LIN {X 0,Y 205.064,Z 329.408,A -85,B 0,C 180,E1 -21802.532,E2 -21802.532} C_VEL
LIN {X 0,Y 207.762,Z 331.827,A -85,B 0,C 180,E1 -21804.481,E2 -21804.481} C_VEL
LIN {X 0,Y 210.172,Z 335.291,A -85,B 0,C 180,E1 -21806.167,E2 -21806.167} C_VEL
LIN {X 0,Y 211.843,Z 337.01,A -85,B 0,C 180,E1 -21807.207,E2 -21807.207} C_VEL
LIN {X 0,Y 214.618,Z 340.729,A -85,B 0,C 180,E1 -21808.883,E2 -21808.883} C_VEL
LIN {X 0,Y 216.211,Z 342.811,A -85,B 0,C 180,E1 -21809.784,E2 -21809.784} C_VEL
LIN {X 0,Y 219.819,Z 347.623,A -85,B 0,C 180,E1 -21811.698,E2 -21811.698} C_VEL
LIN {X 0,Y 224.599,Z 354.224,A -85,B 0,C 180,E1 -21814.01,E2 -21814.01} C_VEL
LIN {X 0,Y 231.76,Z 365.241,A -85,B 0,C 180,E1 -21817.132,E2 -21817.132} C_VEL
LIN {X 0,Y 239.139,Z 377.762,A -85,B 0,C 180,E1 -21820.005,E2 -21820.005} C_VEL
LIN {X 0,Y 243.057,Z 385.535,A -85,B 0,C 180,E1 -21821.444,E2 -21821.444} C_VEL
LIN {X 0,Y 244.176,Z 388.149,A -85,B 0,C 180,E1 -21821.856,E2 -21821.856} C_VEL
LIN {X 0,Y 238.992,Z 467.481,A -85,B 0,C 180,E1 -21823.985,E2 -21823.985} C_VEL
LIN {X 0,Y 237.015,Z 483.086,A -85,B 0,C 180,E1 -21824.632,E2 -21824.632} C_VEL
LIN {X 0,Y 234.342,Z 498.666,A -85,B 0,C 180,E1 -21825.643,E2 -21825.643} C_VEL
LIN {X 0,Y 230.951,Z 513.459,A -85,B 0,C 180,E1 -21826.943,E2 -21826.943} C_VEL
LIN {X 0,Y 227.125,Z 527.553,A -85,B 0,C 180,E1 -21828.594,E2 -21828.594} C_VEL
LIN {X 0,Y 222.938,Z 539.758,A -85,B 0,C 180,E1 -21830.331,E2 -21830.331} C_VEL
LIN {X 0,Y 218.747,Z 551.094,A -85,B 0,C 180,E1 -21832.38,E2 -21832.38} C_VEL
LIN {X 0,Y 213.85,Z 562.546,A -85,B 0,C 180,E1 -21834.893,E2 -21834.893} C_VEL
LIN {X 0,Y 210.165,Z 571.106,A -85,B 0,C 180,E1 -21837.245,E2 -21837.245} C_VEL
LIN {X 0,Y 205.664,Z 580.387,A -85,B 0,C 180,E1 -21840.298,E2 -21840.298} C_VEL
LIN {X 0,Y 201.657,Z 588.46,A -85,B 0,C 180,E1 -21843.619,E2 -21843.619} C_VEL
LIN {X 0,Y 197.889,Z 595.794,A -85,B 0,C 180,E1 -21847.427,E2 -21847.427} C_VEL
LIN {X 0,Y 195.175,Z 601.274,A -85,B 0,C 180,E1 -21851.091,E2 -21851.091} C_VEL
LIN {X 0,Y 192.884,Z 606.023,A -85,B 0,C 180,E1 -21855.224,E2 -21855.224} C_VEL
LIN {X 0,Y 191.454,Z 609.492,A -85,B 0,C 180,E1 -21859.424,E2 -21859.424} C_VEL
LIN {X 0,Y 190.598,Z 611.782,A -85,B 0,C 180,E1 -21863.649,E2 -21863.649} C_VEL
LIN {X 0,Y 190.279,Z 612.946,A -85,B 0,C 180,E1 -21867.883,E2 -21867.883} C_VEL
LIN {X 0,Y 190.301,Z 613.099,A -85,B 0,C 180,E1 -21870,E2 -21870} C_VEL
LIN {X 0,Y 190.444,Z 612.387,A -85,B 0,C 180,E1 -21874.869,E2 -21874.869} C_VEL
LIN {X 0,Y 190.924,Z 610.864,A -85,B 0,C 180,E1 -21878.467,E2 -21878.467} C_VEL
LIN {X 0,Y 192.015,Z 608.037,A -85,B 0,C 180,E1 -21882.686,E2 -21882.686} C_VEL
LIN {X 0,Y 193.838,Z 603.984,A -85,B 0,C 180,E1 -21886.861,E2 -21886.861} C_VEL
LIN {X 0,Y 196.543,Z 598.603,A -85,B 0,C 180,E1 -21890.951,E2 -21890.951} C_VEL
LIN {X 0,Y 199.996,Z 591.742,A -85,B 0,C 180,E1 -21894.941,E2 -21894.941} C_VEL
LIN {X 0,Y 204.381,Z 583.169,A -85,B 0,C 180,E1 -21898.777,E2 -21898.777} C_VEL
LIN {X 0,Y 208.242,Z 575.457,A -85,B 0,C 180,E1 -21901.54,E2 -21901.54} C_VEL
LIN {X 0,Y 212.266,Z 566.382,A -85,B 0,C 180,E1 -21904.253,E2 -21904.253} C_VEL
LIN {X 0,Y 216.975,Z 555.662,A -85,B 0,C 180,E1 -21906.814,E2 -21906.814} C_VEL
LIN {X 0,Y 221.541,Z 543.958,A -85,B 0,C 180,E1 -21909.086,E2 -21909.086} C_VEL
LIN {X 0,Y 226.047,Z 531.167,A -85,B 0,C 180,E1 -21911.054,E2 -21911.054} C_VEL
LIN {X 0,Y 229.823,Z 518.202,A -85,B 0,C 180,E1 -21912.678,E2 -21912.678} C_VEL
LIN {X 0,Y 233.225,Z 504.404,A -85,B 0,C 180,E1 -21914.023,E2 -21914.023} C_VEL
LIN {X 0,Y 236.063,Z 490.138,A -85,B 0,C 180,E1 -21915.072,E2 -21915.072} C_VEL
LIN {X 0,Y 238.303,Z 474.681,A -85,B 0,C 180,E1 -21915.883,E2 -21915.883} C_VEL
LIN {X 0,Y 239.804,Z 458.248,A -85,B 0,C 180,E1 -21916.42,E2 -21916.42} C_VEL
LIN {X 0,Y 244.227,Z 389.062,A -85,B 0,C 180,E1 -21918.255,E2 -21918.255} C_VEL
LIN {X 0,Y 244.113,Z 387.715,A -85,B 0,C 180,E1 -21918.344,E2 -21918.344} C_VEL
LIN {X 0,Y 240.439,Z 379.995,A -85,B 0,C 180,E1 -21919.693,E2 -21919.693} C_VEL
LIN {X 0,Y 233.33,Z 367.712,A -85,B 0,C 180,E1 -21922.417,E2 -21922.417} C_VEL
LIN {X 0,Y 227.065,Z 357.85,A -85,B 0,C 180,E1 -21925.068,E2 -21925.068} C_VEL
LIN {X 0,Y 220.857,Z 348.999,A -85,B 0,C 180,E1 -21927.993,E2 -21927.993} C_VEL
LIN {X 0,Y 217.765,Z 344.83,A -85,B 0,C 180,E1 -21929.595,E2 -21929.595} C_VEL
LIN {X 0,Y 214.67,Z 340.711,A -85,B 0,C 180,E1 -21931.326,E2 -21931.326} C_VEL
LIN {X 0,Y 211.839,Z 336.9,A -85,B 0,C 180,E1 -21933.049,E2 -21933.049} C_VEL
LIN {X 0,Y 208.603,Z 333.276,A -85,B 0,C 180,E1 -21935.16,E2 -21935.16} C_VEL
LIN {X 0,Y 207.462,Z 331.386,A -85,B 0,C 180,E1 -21936.014,E2 -21936.014} C_VEL
LIN {X 0,Y 204.824,Z 329.086,A -85,B 0,C 180,E1 -21937.957,E2 -21937.957} C_VEL
LIN {X 0,Y 202.834,Z 325.858,A -85,B 0,C 180,E1 -21939.727,E2 -21939.727} C_VEL
LIN {X 0,Y 200.217,Z 323.977,A -85,B 0,C 180,E1 -21942.102,E2 -21942.102} C_VEL
LIN {X 0,Y 198.471,Z 321.018,A -85,B 0,C 180,E1 -21944.137,E2 -21944.137} C_VEL
LIN {X 0,Y 198.165,Z 320.138,A -85,B 0,C 180,E1 -21944.574,E2 -21944.574} C_VEL
LIN {X 0,Y 195.141,Z 318.477,A -85,B 0,C 180,E1 -21948.575,E2 -21948.575} C_VEL
LIN {X 0,Y 193.081,Z 314.79,A -85,B 0,C 180,E1 -21953.337,E2 -21953.337} C_VEL
LIN {X 0,Y 192.959,Z 314.068,A -85,B 0,C 180,E1 -21953.989,E2 -21953.989} C_VEL
LIN {X 0,Y 193.229,Z 314.042,A -85,B 0,C 180,E1 -21957.915,E2 -21957.915} C_VEL
LIN {X 0,Y 193.424,Z 314.001,A -85,B 0,C 180,E1 -21960,E2 -21960} C_VEL
LIN {X 0,Y 192.944,Z 314.063,A -85,B 0,C 180,E1 -21965.225,E2 -21965.225} C_VEL
LIN {X 0,Y 193.015,Z 314.43,A -85,B 0,C 180,E1 -21966.009,E2 -21966.009} C_VEL
LIN {X 0,Y 194.229,Z 317.306,A -85,B 0,C 180,E1 -21969.371,E2 -21969.371} C_VEL
LIN {X 0,Y 196.77,Z 319.638,A -85,B 0,C 180,E1 -21973.424,E2 -21973.424} C_VEL
LIN {X 0,Y 198.273,Z 320.416,A -85,B 0,C 180,E1 -21975.22,E2 -21975.22} C_VEL
LIN {X 0,Y 199.493,Z 323.041,A -85,B 0,C 180,E1 -21976.765,E2 -21976.765} C_VEL
LIN {X 0,Y 201.814,Z 325.346,A -85,B 0,C 180,E1 -21979.055,E2 -21979.055} C_VEL
LIN {X 0,Y 203.126,Z 326.222,A -85,B 0,C 180,E1 -21980.176,E2 -21980.176} C_VEL
LIN {X 0,Y 205.214,Z 329.557,A -85,B 0,C 180,E1 -21981.998,E2 -21981.998} C_VEL
LIN {X 0,Y 207.808,Z 331.89,A -85,B 0,C 180,E1 -21983.886,E2 -21983.886} C_VEL
LIN {X 0,Y 210.036,Z 335.119,A -85,B 0,C 180,E1 -21985.464,E2 -21985.464} C_VEL
LIN {X 0,Y 211.903,Z 337.082,A -85,B 0,C 180,E1 -21986.64,E2 -21986.64} C_VEL
LIN {X 0,Y 214.888,Z 340.978,A -85,B 0,C 180,E1 -21988.442,E2 -21988.442} C_VEL
LIN {X 0,Y 219.269,Z 347.018,A -85,B 0,C 180,E1 -21990.852,E2 -21990.852} C_VEL
LIN {X 0,Y 225.018,Z 356.403,A -85,B 0,C 180,E1 -21993.735,E2 -21993.735} C_VEL
LIN {X 0,Y 231.913,Z 369.003,A -85,B 0,C 180,E1 -21996.831,E2 -21996.831} C_VEL
LIN {X 0,Y 233.301,Z 371.742,A -85,B 0,C 180,E1 -21997.416,E2 -21997.416} C_VEL
LIN {X 0,Y 234.372,Z 374.955,A -85,B 0,C 180,E1 -21997.912,E2 -21997.912} C_VEL
LIN {X 0,Y 235.026,Z 381.291,A -85,B 0,C 180,E1 -21998.42,E2 -21998.42} C_VEL
LIN {X 0,Y 235.535,Z 387.812,A -85,B 0,C 180,E1 -21998.885,E2 -21998.885} C_VEL
LIN {X 0,Y 236.429,Z 391.32,A -85,B 0,C 180,E1 -21999.315,E2 -21999.315} C_VEL
LIN {X 0,Y 239.07,Z 397.805,A -85,B 0,C 180,E1 -22000.372,E2 -22000.372} C_VEL
LIN {X 0,Y 233.646,Z 477.533,A -85,B 0,C 180,E1 -22002.529,E2 -22002.529} C_VEL
LIN {X 0,Y 231.44,Z 493.66,A -85,B 0,C 180,E1 -22003.216,E2 -22003.216} C_VEL
LIN {X 0,Y 228.735,Z 507.71,A -85,B 0,C 180,E1 -22004.095,E2 -22004.095} C_VEL
LIN {X 0,Y 225.53,Z 520.652,A -85,B 0,C 180,E1 -22005.169,E2 -22005.169} C_VEL
LIN {X 0,Y 221.439,Z 534.513,A -85,B 0,C 180,E1 -22006.662,E2 -22006.662} C_VEL
LIN {X 0,Y 217.053,Z 547.492,A -85,B 0,C 180,E1 -22008.479,E2 -22008.479} C_VEL
LIN {X 0,Y 211.997,Z 560.073,A -85,B 0,C 180,E1 -22010.654,E2 -22010.654} C_VEL
LIN {X 0,Y 207.278,Z 570.843,A -85,B 0,C 180,E1 -22013,E2 -22013} C_VEL
LIN {X 0,Y 202.594,Z 580.815,A -85,B 0,C 180,E1 -22015.688,E2 -22015.688} C_VEL
LIN {X 0,Y 197.765,Z 590.579,A -85,B 0,C 180,E1 -22018.984,E2 -22018.984} C_VEL
LIN {X 0,Y 194.203,Z 597.652,A -85,B 0,C 180,E1 -22021.937,E2 -22021.937} C_VEL
LIN {X 0,Y 190.107,Z 605.481,A -85,B 0,C 180,E1 -22026.006,E2 -22026.006} C_VEL
LIN {X 0,Y 187.03,Z 611.719,A -85,B 0,C 180,E1 -22030.234,E2 -22030.234} C_VEL
LIN {X 0,Y 184.914,Z 616.552,A -85,B 0,C 180,E1 -22034.571,E2 -22034.571} C_VEL
LIN {X 0,Y 183.591,Z 620.099,A -85,B 0,C 180,E1 -22038.966,E2 -22038.966} C_VEL
LIN {X 0,Y 183.085,Z 622.44,A -85,B 0,C 180,E1 -22043.387,E2 -22043.387} C_VEL
LIN {X 0,Y 183.04,Z 623.62,A -85,B 0,C 180,E1 -22047.8,E2 -22047.8} C_VEL
LIN {X 0,Y 183.168,Z 623.778,A -85,B 0,C 180,E1 -22050,E2 -22050} C_VEL
LIN {X 0,Y 182.976,Z 623.157,A -85,B 0,C 180,E1 -22054.406,E2 -22054.406} C_VEL
LIN {X 0,Y 183.225,Z 621.38,A -85,B 0,C 180,E1 -22058.825,E2 -22058.825} C_VEL
LIN {X 0,Y 184.092,Z 618.428,A -85,B 0,C 180,E1 -22063.241,E2 -22063.241} C_VEL
LIN {X 0,Y 185.812,Z 614.236,A -85,B 0,C 180,E1 -22067.612,E2 -22067.612} C_VEL
LIN {X 0,Y 188.423,Z 608.695,A -85,B 0,C 180,E1 -22071.9,E2 -22071.9} C_VEL
LIN {X 0,Y 192.033,Z 601.659,A -85,B 0,C 180,E1 -22076.05,E2 -22076.05} C_VEL
LIN {X 0,Y 196.637,Z 592.918,A -85,B 0,C 180,E1 -22080.024,E2 -22080.024} C_VEL
LIN {X 0,Y 201.16,Z 583.633,A -85,B 0,C 180,E1 -22083.383,E2 -22083.383} C_VEL
LIN {X 0,Y 205.675,Z 574.202,A -85,B 0,C 180,E1 -22086.116,E2 -22086.116} C_VEL
LIN {X 0,Y 210.659,Z 563.005,A -85,B 0,C 180,E1 -22088.72,E2 -22088.72} C_VEL
LIN {X 0,Y 215.673,Z 550.847,A -85,B 0,C 180,E1 -22090.951,E2 -22090.951} C_VEL
LIN {X 0,Y 220.371,Z 537.398,A -85,B 0,C 180,E1 -22092.942,E2 -22092.942} C_VEL
LIN {X 0,Y 224.461,Z 523.999,A -85,B 0,C 180,E1 -22094.471,E2 -22094.471} C_VEL
LIN {X 0,Y 227.932,Z 510.63,A -85,B 0,C 180,E1 -22095.638,E2 -22095.638} C_VEL
LIN {X 0,Y 230.901,Z 495.994,A -85,B 0,C 180,E1 -22096.608,E2 -22096.608} C_VEL
LIN {X 0,Y 233.061,Z 481.047,A -85,B 0,C 180,E1 -22097.308,E2 -22097.308} C_VEL
LIN {X 0,Y 234.774,Z 461.127,A -85,B 0,C 180,E1 -22097.886,E2 -22097.886} C_VEL
LIN {X 0,Y 238.926,Z 397.592,A -85,B 0,C 180,E1 -22099.599,E2 -22099.599} C_VEL
LIN {X 0,Y 233.213,Z 384.116,A -85,B 0,C 180,E1 -22101.915,E2 -22101.915} C_VEL
LIN {X 0,Y 227.596,Z 372.514,A -85,B 0,C 180,E1 -22104.349,E2 -22104.349} C_VEL
LIN {X 0,Y 221.336,Z 360.866,A -85,B 0,C 180,E1 -22107.331,E2 -22107.331} C_VEL
LIN {X 0,Y 215.492,Z 351.159,A -85,B 0,C 180,E1 -22110.449,E2 -22110.449} C_VEL
LIN {X 0,Y 212.534,Z 347.151,A -85,B 0,C 180,E1 -22112.155,E2 -22112.155} C_VEL
LIN {X 0,Y 208.878,Z 342.408,A -85,B 0,C 180,E1 -22114.463,E2 -22114.463} C_VEL
LIN {X 0,Y 206.271,Z 339.136,A -85,B 0,C 180,E1 -22116.281,E2 -22116.281} C_VEL
LIN {X 0,Y 205.347,Z 337.852,A -85,B 0,C 180,E1 -22116.979,E2 -22116.979} C_VEL
LIN {X 0,Y 202.664,Z 335.074,A -85,B 0,C 180,E1 -22119.079,E2 -22119.079} C_VEL
LIN {X 0,Y 201.289,Z 332.655,A -85,B 0,C 180,E1 -22120.363,E2 -22120.363} C_VEL
LIN {X 0,Y 198.707,Z 330.594,A -85,B 0,C 180,E1 -22122.781,E2 -22122.781} C_VEL
LIN {X 0,Y 196.913,Z 327.525,A -85,B 0,C 180,E1 -22124.938,E2 -22124.938} C_VEL
LIN {X 0,Y 196.473,Z 326.921,A -85,B 0,C 180,E1 -22125.499,E2 -22125.499} C_VEL
LIN {X 0,Y 193.732,Z 325.021,A -85,B 0,C 180,E1 -22129.352,E2 -22129.352} C_VEL
LIN {X 0,Y 192.022,Z 321.595,A -85,B 0,C 180,E1 -22133.433,E2 -22133.433} C_VEL
LIN {X 0,Y 191.795,Z 321.046,A -85,B 0,C 180,E1 -22134.217,E2 -22134.217} C_VEL
LIN {X 0,Y 190.798,Z 320.606,A -85,B 0,C 180,E1 -22140,E2 -22140} C_VEL
LIN {X 0,Y 191.99,Z 321.277,A -85,B 0,C 180,E1 -22146.833,E2 -22146.833} C_VEL
LIN {X 0,Y 193.151,Z 324.251,A -85,B 0,C 180,E1 -22149.995,E2 -22149.995} C_VEL
LIN {X 0,Y 195.514,Z 326.526,A -85,B 0,C 180,E1 -22153.777,E2 -22153.777} C_VEL
LIN {X 0,Y 196.813,Z 327.23,A -85,B 0,C 180,E1 -22155.362,E2 -22155.362} C_VEL
LIN {X 0,Y 198.669,Z 330.618,A -85,B 0,C 180,E1 -22157.635,E2 -22157.635} C_VEL
LIN {X 0,Y 201.497,Z 332.983,A -85,B 0,C 180,E1 -22160.28,E2 -22160.28} C_VEL
LIN {X 0,Y 203.636,Z 336.307,A -85,B 0,C 180,E1 -22162.178,E2 -22162.178} C_VEL
LIN {X 0,Y 205.865,Z 338.411,A -85,B 0,C 180,E1 -22163.85,E2 -22163.85} C_VEL
LIN {X 0,Y 208.649,Z 342.169,A -85,B 0,C 180,E1 -22165.835,E2 -22165.835} C_VEL
LIN {X 0,Y 209.923,Z 343.725,A -85,B 0,C 180,E1 -22166.669,E2 -22166.669} C_VEL
LIN {X 0,Y 213.841,Z 348.947,A -85,B 0,C 180,E1 -22169.065,E2 -22169.065} C_VEL
LIN {X 0,Y 217.656,Z 354.201,A -85,B 0,C 180,E1 -22171.171,E2 -22171.171} C_VEL
LIN {X 0,Y 222.226,Z 360.833,A -85,B 0,C 180,E1 -22173.468,E2 -22173.468} C_VEL
LIN {X 0,Y 228.382,Z 370.38,A -85,B 0,C 180,E1 -22176.258,E2 -22176.258} C_VEL
LIN {X 0,Y 235.566,Z 382.867,A -85,B 0,C 180,E1 -22179.192,E2 -22179.192} C_VEL
LIN {X 0,Y 239,Z 389.847,A -85,B 0,C 180,E1 -22180.518,E2 -22180.518} C_VEL
LIN {X 0,Y 239.32,Z 390.603,A -85,B 0,C 180,E1 -22180.642,E2 -22180.642} C_VEL
LIN {X 0,Y 234.137,Z 467.703,A -85,B 0,C 180,E1 -22182.739,E2 -22182.739} C_VEL
LIN {X 0,Y 232.088,Z 483.301,A -85,B 0,C 180,E1 -22183.387,E2 -22183.387} C_VEL
LIN {X 0,Y 229.335,Z 498.877,A -85,B 0,C 180,E1 -22184.407,E2 -22184.407} C_VEL
LIN {X 0,Y 225.854,Z 513.542,A -85,B 0,C 180,E1 -22185.701,E2 -22185.701} C_VEL
LIN {X 0,Y 221.852,Z 527.761,A -85,B 0,C 180,E1 -22187.381,E2 -22187.381} C_VEL
LIN {X 0,Y 217.062,Z 541.206,A -85,B 0,C 180,E1 -22189.339,E2 -22189.339} C_VEL
LIN {X 0,Y 212.31,Z 553.401,A -85,B 0,C 180,E1 -22191.636,E2 -22191.636} C_VEL
LIN {X 0,Y 207.283,Z 564.518,A -85,B 0,C 180,E1 -22194.208,E2 -22194.208} C_VEL
LIN {X 0,Y 202.289,Z 575.296,A -85,B 0,C 180,E1 -22197.419,E2 -22197.419} C_VEL
LIN {X 0,Y 197.641,Z 584.25,A -85,B 0,C 180,E1 -22200.73,E2 -22200.73} C_VEL
LIN {X 0,Y 193.632,Z 591.665,A -85,B 0,C 180,E1 -22204.181,E2 -22204.181} C_VEL
LIN {X 0,Y 189.912,Z 598.589,A -85,B 0,C 180,E1 -22208.281,E2 -22208.281} C_VEL
LIN {X 0,Y 187.069,Z 604.022,A -85,B 0,C 180,E1 -22212.51,E2 -22212.51} C_VEL
LIN {X 0,Y 185.131,Z 608.115,A -85,B 0,C 180,E1 -22216.834,E2 -22216.834} C_VEL
LIN {X 0,Y 183.898,Z 610.985,A -85,B 0,C 180,E1 -22221.207,E2 -22221.207} C_VEL
LIN {X 0,Y 183.308,Z 612.706,A -85,B 0,C 180,E1 -22225.602,E2 -22225.602} C_VEL
LIN {X 0,Y 183.207,Z 613.302,A -85,B 0,C 180,E1 -22230,E2 -22230} C_VEL
LIN {X 0,Y 183.331,Z 612.688,A -85,B 0,C 180,E1 -22234.644,E2 -22234.644} C_VEL
LIN {X 0,Y 183.877,Z 611.067,A -85,B 0,C 180,E1 -22238.794,E2 -22238.794} C_VEL
LIN {X 0,Y 185.081,Z 608.239,A -85,B 0,C 180,E1 -22243.169,E2 -22243.169} C_VEL
LIN {X 0,Y 187.039,Z 604.187,A -85,B 0,C 180,E1 -22247.493,E2 -22247.493} C_VEL
LIN {X 0,Y 189.904,Z 598.805,A -85,B 0,C 180,E1 -22251.72,E2 -22251.72} C_VEL
LIN {X 0,Y 193.545,Z 591.945,A -85,B 0,C 180,E1 -22255.832,E2 -22255.832} C_VEL
LIN {X 0,Y 198.152,Z 583.372,A -85,B 0,C 180,E1 -22259.771,E2 -22259.771} C_VEL
LIN {X 0,Y 202.89,Z 574.25,A -85,B 0,C 180,E1 -22263.063,E2 -22263.063} C_VEL
LIN {X 0,Y 207.213,Z 564.964,A -85,B 0,C 180,E1 -22265.806,E2 -22265.806} C_VEL
LIN {X 0,Y 212.614,Z 552.927,A -85,B 0,C 180,E1 -22268.602,E2 -22268.602} C_VEL
LIN {X 0,Y 217.451,Z 540.634,A -85,B 0,C 180,E1 -22270.879,E2 -22270.879} C_VEL
LIN {X 0,Y 222.157,Z 527.057,A -85,B 0,C 180,E1 -22272.854,E2 -22272.854} C_VEL
LIN {X 0,Y 226.107,Z 513.222,A -85,B 0,C 180,E1 -22274.455,E2 -22274.455} C_VEL
LIN {X 0,Y 229.418,Z 498.939,A -85,B 0,C 180,E1 -22275.729,E2 -22275.729} C_VEL
LIN {X 0,Y 232.276,Z 483.381,A -85,B 0,C 180,E1 -22276.722,E2 -22276.722} C_VEL
LIN {X 0,Y 234.233,Z 467.862,A -85,B 0,C 180,E1 -22277.394,E2 -22277.394} C_VEL
LIN {X 0,Y 239.442,Z 390.666,A -85,B 0,C 180,E1 -22279.49,E2 -22279.49} C_VEL
LIN {X 0,Y 236.263,Z 384.057,A -85,B 0,C 180,E1 -22280.718,E2 -22280.718} C_VEL
LIN {X 0,Y 229.752,Z 372.645,A -85,B 0,C 180,E1 -22283.345,E2 -22283.345} C_VEL
LIN {X 0,Y 224.127,Z 363.557,A -85,B 0,C 180,E1 -22285.844,E2 -22285.844} C_VEL
LIN {X 0,Y 218.282,Z 354.993,A -85,B 0,C 180,E1 -22288.723,E2 -22288.723} C_VEL
LIN {X 0,Y 215.07,Z 350.604,A -85,B 0,C 180,E1 -22290.463,E2 -22290.463} C_VEL
LIN {X 0,Y 212.44,Z 346.967,A -85,B 0,C 180,E1 -22292.007,E2 -22292.007} C_VEL
LIN {X 0,Y 208.965,Z 342.435,A -85,B 0,C 180,E1 -22294.222,E2 -22294.222} C_VEL
LIN {X 0,Y 206.401,Z 339.271,A -85,B 0,C 180,E1 -22296.016,E2 -22296.016} C_VEL
LIN {X 0,Y 205.504,Z 337.913,A -85,B 0,C 180,E1 -22296.707,E2 -22296.707} C_VEL
LIN {X 0,Y 202.835,Z 335.254,A -85,B 0,C 180,E1 -22298.798,E2 -22298.798} C_VEL
LIN {X 0,Y 201.165,Z 332.591,A -85,B 0,C 180,E1 -22300.35,E2 -22300.35} C_VEL
LIN {X 0,Y 198.538,Z 330.382,A -85,B 0,C 180,E1 -22302.889,E2 -22302.889} C_VEL
LIN {X 0,Y 196.823,Z 327.143,A -85,B 0,C 180,E1 -22305.063,E2 -22305.063} C_VEL
LIN {X 0,Y 193.7,Z 324.984,A -85,B 0,C 180,E1 -22309.548,E2 -22309.548} C_VEL
LIN {X 0,Y 192.002,Z 321.331,A -85,B 0,C 180,E1 -22314.091,E2 -22314.091} C_VEL
LIN {X 0,Y 191.119,Z 320.718,A -85,B 0,C 180,E1 -22320,E2 -22320} C_VEL
LIN {X 0,Y 191.999,Z 321.259,A -85,B 0,C 180,E1 -22325.514,E2 -22325.514} C_VEL
LIN {X 0,Y 193.152,Z 324.196,A -85,B 0,C 180,E1 -22328.978,E2 -22328.978} C_VEL
LIN {X 0,Y 195.73,Z 326.63,A -85,B 0,C 180,E1 -22333.232,E2 -22333.232} C_VEL
LIN {X 0,Y 196.881,Z 327.318,A -85,B 0,C 180,E1 -22334.668,E2 -22334.668} C_VEL
LIN {X 0,Y 198.372,Z 330.127,A -85,B 0,C 180,E1 -22336.564,E2 -22336.564} C_VEL
LIN {X 0,Y 200.778,Z 332.406,A -85,B 0,C 180,E1 -22338.958,E2 -22338.958} C_VEL
LIN {X 0,Y 201.542,Z 333.045,A -85,B 0,C 180,E1 -22339.64,E2 -22339.64} C_VEL
LIN {X 0,Y 203.774,Z 336.413,A -85,B 0,C 180,E1 -22341.629,E2 -22341.629} C_VEL
LIN {X 0,Y 205.943,Z 338.467,A -85,B 0,C 180,E1 -22343.267,E2 -22343.267} C_VEL
LIN {X 0,Y 208.584,Z 342.095,A -85,B 0,C 180,E1 -22345.175,E2 -22345.175} C_VEL
LIN {X 0,Y 209.935,Z 343.701,A -85,B 0,C 180,E1 -22346.064,E2 -22346.064} C_VEL
LIN {X 0,Y 213.919,Z 348.983,A -85,B 0,C 180,E1 -22348.516,E2 -22348.516} C_VEL
LIN {X 0,Y 216.726,Z 353.058,A -85,B 0,C 180,E1 -22350.107,E2 -22350.107} C_VEL
LIN {X 0,Y 222.224,Z 362.35,A -85,B 0,C 180,E1 -22352.994,E2 -22352.994} C_VEL
LIN {X 0,Y 228.524,Z 374.162,A -85,B 0,C 180,E1 -22355.959,E2 -22355.959} C_VEL
LIN {X 0,Y 234.286,Z 386.293,A -85,B 0,C 180,E1 -22358.434,E2 -22358.434} C_VEL
LIN {X 0,Y 236.429,Z 391.32,A -85,B 0,C 180,E1 -22359.315,E2 -22359.315} C_VEL
LIN {X 0,Y 236.972,Z 394.195,A -85,B 0,C 180,E1 -22359.608,E2 -22359.608} C_VEL
LIN {X 0,Y 236.608,Z 398.725,A -85,B 0,C 180,E1 -22359.713,E2 -22359.713} C_VEL
LIN {X 0,Y 233.717,Z 411.006,A -85,B 0,C 180,E1 -22359.44,E2 -22359.44} C_VEL
LIN {X 0,Y 233.561,Z 412.418,A -85,B 0,C 180,E1 -22359.461,E2 -22359.461} C_VEL
LIN {X 0,Y 228.918,Z 477.347,A -85,B 0,C 180,E1 -22361.223,E2 -22361.223} C_VEL
LIN {X 0,Y 226.636,Z 493.466,A -85,B 0,C 180,E1 -22361.908,E2 -22361.908} C_VEL
LIN {X 0,Y 223.851,Z 507.515,A -85,B 0,C 180,E1 -22362.789,E2 -22362.789} C_VEL
LIN {X 0,Y 220.006,Z 522.439,A -85,B 0,C 180,E1 -22364.05,E2 -22364.05} C_VEL
LIN {X 0,Y 215.789,Z 535.9,A -85,B 0,C 180,E1 -22365.558,E2 -22365.558} C_VEL
LIN {X 0,Y 211.205,Z 548.802,A -85,B 0,C 180,E1 -22367.437,E2 -22367.437} C_VEL
LIN {X 0,Y 205.595,Z 562.017,A -85,B 0,C 180,E1 -22369.819,E2 -22369.819} C_VEL
LIN {X 0,Y 199.921,Z 574.194,A -85,B 0,C 180,E1 -22372.671,E2 -22372.671} C_VEL
LIN {X 0,Y 194.443,Z 585.034,A -85,B 0,C 180,E1 -22375.929,E2 -22375.929} C_VEL
LIN {X 0,Y 189.797,Z 594.076,A -85,B 0,C 180,E1 -22379.394,E2 -22379.394} C_VEL
LIN {X 0,Y 185.573,Z 601.575,A -85,B 0,C 180,E1 -22382.97,E2 -22382.97} C_VEL
LIN {X 0,Y 181.793,Z 608.581,A -85,B 0,C 180,E1 -22387.258,E2 -22387.258} C_VEL
LIN {X 0,Y 179.041,Z 614.099,A -85,B 0,C 180,E1 -22391.698,E2 -22391.698} C_VEL
LIN {X 0,Y 177.132,Z 618.275,A -85,B 0,C 180,E1 -22396.228,E2 -22396.228} C_VEL
LIN {X 0,Y 176.212,Z 621.214,A -85,B 0,C 180,E1 -22400.82,E2 -22400.82} C_VEL
LIN {X 0,Y 175.882,Z 622.969,A -85,B 0,C 180,E1 -22405.416,E2 -22405.416} C_VEL
LIN {X 0,Y 176.075,Z 623.575,A -85,B 0,C 180,E1 -22410,E2 -22410} C_VEL
LIN {X 0,Y 175.876,Z 622.953,A -85,B 0,C 180,E1 -22414.584,E2 -22414.584} C_VEL
LIN {X 0,Y 176.182,Z 621.176,A -85,B 0,C 180,E1 -22419.181,E2 -22419.181} C_VEL
LIN {X 0,Y 177.125,Z 618.222,A -85,B 0,C 180,E1 -22423.772,E2 -22423.772} C_VEL
LIN {X 0,Y 178.993,Z 614.03,A -85,B 0,C 180,E1 -22428.307,E2 -22428.307} C_VEL
LIN {X 0,Y 181.779,Z 608.488,A -85,B 0,C 180,E1 -22432.744,E2 -22432.744} C_VEL
LIN {X 0,Y 185.592,Z 601.452,A -85,B 0,C 180,E1 -22437.027,E2 -22437.027} C_VEL
LIN {X 0,Y 189.824,Z 593.938,A -85,B 0,C 180,E1 -22440.601,E2 -22440.601} C_VEL
LIN {X 0,Y 194.48,Z 584.879,A -85,B 0,C 180,E1 -22444.062,E2 -22444.062} C_VEL
LIN {X 0,Y 199.936,Z 573.995,A -85,B 0,C 180,E1 -22447.325,E2 -22447.325} C_VEL
LIN {X 0,Y 205.129,Z 562.797,A -85,B 0,C 180,E1 -22449.97,E2 -22449.97} C_VEL
LIN {X 0,Y 210.714,Z 549.735,A -85,B 0,C 180,E1 -22452.375,E2 -22452.375} C_VEL
LIN {X 0,Y 215.272,Z 537.043,A -85,B 0,C 180,E1 -22454.252,E2 -22454.252} C_VEL
LIN {X 0,Y 219.434,Z 523.789,A -85,B 0,C 180,E1 -22455.775,E2 -22455.775} C_VEL
LIN {X 0,Y 223.024,Z 510.42,A -85,B 0,C 180,E1 -22456.943,E2 -22456.943} C_VEL
LIN {X 0,Y 226.09,Z 495.782,A -85,B 0,C 180,E1 -22457.913,E2 -22457.913} C_VEL
LIN {X 0,Y 228.313,Z 480.831,A -85,B 0,C 180,E1 -22458.616,E2 -22458.616} C_VEL
LIN {X 0,Y 230.079,Z 460.902,A -85,B 0,C 180,E1 -22459.196,E2 -22459.196} C_VEL
LIN {X 0,Y 234.172,Z 400.03,A -85,B 0,C 180,E1 -22460.859,E2 -22460.859} C_VEL
LIN {X 0,Y 228.729,Z 387.124,A -85,B 0,C 180,E1 -22463.206,E2 -22463.206} C_VEL
LIN {X 0,Y 223.858,Z 376.859,A -85,B 0,C 180,E1 -22465.454,E2 -22465.454} C_VEL
LIN {X 0,Y 218.205,Z 366.075,A -85,B 0,C 180,E1 -22468.305,E2 -22468.305} C_VEL
LIN {X 0,Y 212.932,Z 357.043,A -85,B 0,C 180,E1 -22471.272,E2 -22471.272} C_VEL
LIN {X 0,Y 210.014,Z 353.029,A -85,B 0,C 180,E1 -22473.039,E2 -22473.039} C_VEL
LIN {X 0,Y 206.89,Z 348.835,A -85,B 0,C 180,E1 -22475.108,E2 -22475.108} C_VEL
LIN {X 0,Y 204.048,Z 345.033,A -85,B 0,C 180,E1 -22477.202,E2 -22477.202} C_VEL
LIN {X 0,Y 200.618,Z 341.069,A -85,B 0,C 180,E1 -22480.028,E2 -22480.028} C_VEL
LIN {X 0,Y 199.633,Z 339.332,A -85,B 0,C 180,E1 -22480.996,E2 -22480.996} C_VEL
LIN {X 0,Y 197.061,Z 337.018,A -85,B 0,C 180,E1 -22483.556,E2 -22483.556} C_VEL
LIN {X 0,Y 195.213,Z 333.811,A -85,B 0,C 180,E1 -22485.936,E2 -22485.936} C_VEL
LIN {X 0,Y 192.63,Z 331.89,A -85,B 0,C 180,E1 -22489.734,E2 -22489.734} C_VEL
LIN {X 0,Y 190.987,Z 328.438,A -85,B 0,C 180,E1 -22493.927,E2 -22493.927} C_VEL
LIN {X 0,Y 190.758,Z 328.095,A -85,B 0,C 180,E1 -22494.715,E2 -22494.715} C_VEL
LIN {X 0,Y 189.935,Z 327.636,A -85,B 0,C 180,E1 -22500,E2 -22500} C_VEL
LIN {X 0,Y 190.994,Z 328.307,A -85,B 0,C 180,E1 -22506.496,E2 -22506.496} C_VEL
LIN {X 0,Y 192.246,Z 331.449,A -85,B 0,C 180,E1 -22509.98,E2 -22509.98} C_VEL
LIN {X 0,Y 194.476,Z 333.519,A -85,B 0,C 180,E1 -22513.586,E2 -22513.586} C_VEL
LIN {X 0,Y 195.512,Z 334.198,A -85,B 0,C 180,E1 -22514.907,E2 -22514.907} C_VEL
LIN {X 0,Y 197.348,Z 337.444,A -85,B 0,C 180,E1 -22517.219,E2 -22517.219} C_VEL
LIN {X 0,Y 199.945,Z 339.786,A -85,B 0,C 180,E1 -22519.754,E2 -22519.754} C_VEL
LIN {X 0,Y 202.241,Z 343.19,A -85,B 0,C 180,E1 -22521.836,E2 -22521.836} C_VEL
LIN {X 0,Y 204.074,Z 345.048,A -85,B 0,C 180,E1 -22523.264,E2 -22523.264} C_VEL
LIN {X 0,Y 206.928,Z 348.839,A -85,B 0,C 180,E1 -22525.362,E2 -22525.362} C_VEL
LIN {X 0,Y 211.37,Z 354.878,A -85,B 0,C 180,E1 -22528.247,E2 -22528.247} C_VEL
LIN {X 0,Y 216.592,Z 362.235,A -85,B 0,C 180,E1 -22531.209,E2 -22531.209} C_VEL
LIN {X 0,Y 223.365,Z 372.755,A -85,B 0,C 180,E1 -22534.582,E2 -22534.582} C_VEL
LIN {X 0,Y 230.628,Z 385.38,A -85,B 0,C 180,E1 -22537.776,E2 -22537.776} C_VEL
LIN {X 0,Y 234.591,Z 393.21,A -85,B 0,C 180,E1 -22539.39,E2 -22539.39} C_VEL
LIN {X 0,Y 229.394,Z 467.968,A -85,B 0,C 180,E1 -22541.444,E2 -22541.444} C_VEL
LIN {X 0,Y 227.291,Z 483.515,A -85,B 0,C 180,E1 -22542.092,E2 -22542.092} C_VEL
LIN {X 0,Y 224.425,Z 499.088,A -85,B 0,C 180,E1 -22543.112,E2 -22543.112} C_VEL
LIN {X 0,Y 220.91,Z 513.464,A -85,B 0,C 180,E1 -22544.387,E2 -22544.387} C_VEL
LIN {X 0,Y 216.675,Z 527.969,A -85,B 0,C 180,E1 -22546.109,E2 -22546.109} C_VEL
LIN {X 0,Y 211.727,Z 541.413,A -85,B 0,C 180,E1 -22548.087,E2 -22548.087} C_VEL
LIN {X 0,Y 206.776,Z 553.608,A -85,B 0,C 180,E1 -22550.412,E2 -22550.412} C_VEL
LIN {X 0,Y 201.558,Z 564.724,A -85,B 0,C 180,E1 -22553.025,E2 -22553.025} C_VEL
LIN {X 0,Y 197.763,Z 572.583,A -85,B 0,C 180,E1 -22555.349,E2 -22555.349} C_VEL
LIN {X 0,Y 192.731,Z 582.021,A -85,B 0,C 180,E1 -22558.694,E2 -22558.694} C_VEL
LIN {X 0,Y 187.806,Z 590.871,A -85,B 0,C 180,E1 -22562.716,E2 -22562.716} C_VEL
LIN {X 0,Y 184.35,Z 596.923,A -85,B 0,C 180,E1 -22566.2,E2 -22566.2} C_VEL
LIN {X 0,Y 181.012,Z 602.998,A -85,B 0,C 180,E1 -22570.73,E2 -22570.73} C_VEL
LIN {X 0,Y 179.093,Z 606.433,A -85,B 0,C 180,E1 -22574.057,E2 -22574.057} C_VEL
LIN {X 0,Y 177.456,Z 609.901,A -85,B 0,C 180,E1 -22578.579,E2 -22578.579} C_VEL
LIN {X 0,Y 176.468,Z 612.19,A -85,B 0,C 180,E1 -22583.138,E2 -22583.138} C_VEL
LIN {X 0,Y 176.106,Z 613.351,A -85,B 0,C 180,E1 -22587.713,E2 -22587.713} C_VEL
LIN {X 0,Y 176.116,Z 613.505,A -85,B 0,C 180,E1 -22590,E2 -22590} C_VEL
LIN {X 0,Y 176.226,Z 612.943,A -85,B 0,C 180,E1 -22594.575,E2 -22594.575} C_VEL
LIN {X 0,Y 176.845,Z 611.27,A -85,B 0,C 180,E1 -22599.147,E2 -22599.147} C_VEL
LIN {X 0,Y 178.129,Z 608.443,A -85,B 0,C 180,E1 -22603.693,E2 -22603.693} C_VEL
LIN {X 0,Y 180.269,Z 604.389,A -85,B 0,C 180,E1 -22608.173,E2 -22608.173} C_VEL
LIN {X 0,Y 183.307,Z 599.007,A -85,B 0,C 180,E1 -22612.544,E2 -22612.544} C_VEL
LIN {X 0,Y 187.167,Z 592.147,A -85,B 0,C 180,E1 -22616.781,E2 -22616.781} C_VEL
LIN {X 0,Y 191.997,Z 583.573,A -85,B 0,C 180,E1 -22620.827,E2 -22620.827} C_VEL
LIN {X 0,Y 196.931,Z 574.452,A -85,B 0,C 180,E1 -22624.199,E2 -22624.199} C_VEL
LIN {X 0,Y 200.669,Z 566.783,A -85,B 0,C 180,E1 -22626.539,E2 -22626.539} C_VEL
LIN {X 0,Y 205.757,Z 556.063,A -85,B 0,C 180,E1 -22629.189,E2 -22629.189} C_VEL
LIN {X 0,Y 210.679,Z 544.357,A -85,B 0,C 180,E1 -22631.528,E2 -22631.528} C_VEL
LIN {X 0,Y 215.542,Z 531.563,A -85,B 0,C 180,E1 -22633.534,E2 -22633.534} C_VEL
LIN {X 0,Y 219.922,Z 517.539,A -85,B 0,C 180,E1 -22635.3,E2 -22635.3} C_VEL
LIN {X 0,Y 223.755,Z 502.541,A -85,B 0,C 180,E1 -22636.743,E2 -22636.743} C_VEL
LIN {X 0,Y 226.785,Z 487.482,A -85,B 0,C 180,E1 -22637.802,E2 -22637.802} C_VEL
LIN {X 0,Y 228.936,Z 472.78,A -85,B 0,C 180,E1 -22638.523,E2 -22638.523} C_VEL
LIN {X 0,Y 230.643,Z 453.245,A -85,B 0,C 180,E1 -22639.117,E2 -22639.117} C_VEL
LIN {X 0,Y 234.689,Z 393.183,A -85,B 0,C 180,E1 -22640.757,E2 -22640.757} C_VEL
LIN {X 0,Y 229.645,Z 383.442,A -85,B 0,C 180,E1 -22642.827,E2 -22642.827} C_VEL
LIN {X 0,Y 222.687,Z 371.596,A -85,B 0,C 180,E1 -22645.939,E2 -22645.939} C_VEL
LIN {X 0,Y 216.334,Z 361.755,A -85,B 0,C 180,E1 -22649.155,E2 -22649.155} C_VEL
LIN {X 0,Y 210.419,Z 353.421,A -85,B 0,C 180,E1 -22652.594,E2 -22652.594} C_VEL
LIN {X 0,Y 206.867,Z 348.778,A -85,B 0,C 180,E1 -22654.945,E2 -22654.945} C_VEL
LIN {X 0,Y 204.03,Z 344.901,A -85,B 0,C 180,E1 -22657.066,E2 -22657.066} C_VEL
LIN {X 0,Y 200.764,Z 341.21,A -85,B 0,C 180,E1 -22659.776,E2 -22659.776} C_VEL
LIN {X 0,Y 199.791,Z 339.451,A -85,B 0,C 180,E1 -22660.744,E2 -22660.744} C_VEL
LIN {X 0,Y 197.007,Z 336.928,A -85,B 0,C 180,E1 -22663.563,E2 -22663.563} C_VEL
LIN {X 0,Y 195.417,Z 333.905,A -85,B 0,C 180,E1 -22665.685,E2 -22665.685} C_VEL
LIN {X 0,Y 192.721,Z 332.002,A -85,B 0,C 180,E1 -22669.718,E2 -22669.718} C_VEL
LIN {X 0,Y 190.965,Z 328.126,A -85,B 0,C 180,E1 -22674.721,E2 -22674.721} C_VEL
LIN {X 0,Y 190.254,Z 327.765,A -85,B 0,C 180,E1 -22680,E2 -22680} C_VEL
LIN {X 0,Y 191.013,Z 328.283,A -85,B 0,C 180,E1 -22685.145,E2 -22685.145} C_VEL
LIN {X 0,Y 192.895,Z 332.208,A -85,B 0,C 180,E1 -22690.252,E2 -22690.252} C_VEL
LIN {X 0,Y 195.559,Z 334.244,A -85,B 0,C 180,E1 -22694.171,E2 -22694.171} C_VEL
LIN {X 0,Y 197.416,Z 337.445,A -85,B 0,C 180,E1 -22696.547,E2 -22696.547} C_VEL
LIN {X 0,Y 199.987,Z 339.847,A -85,B 0,C 180,E1 -22699.102,E2 -22699.102} C_VEL
LIN {X 0,Y 202.485,Z 343.436,A -85,B 0,C 180,E1 -22701.373,E2 -22701.373} C_VEL
LIN {X 0,Y 204.182,Z 345.187,A -85,B 0,C 180,E1 -22702.704,E2 -22702.704} C_VEL
LIN {X 0,Y 207.2,Z 349.111,A -85,B 0,C 180,E1 -22704.922,E2 -22704.922} C_VEL
LIN {X 0,Y 211.765,Z 355.382,A -85,B 0,C 180,E1 -22707.887,E2 -22707.887} C_VEL
LIN {X 0,Y 214.157,Z 358.988,A -85,B 0,C 180,E1 -22709.307,E2 -22709.307} C_VEL
LIN {X 0,Y 219.079,Z 367.518,A -85,B 0,C 180,E1 -22712.027,E2 -22712.027} C_VEL
LIN {X 0,Y 225.292,Z 379.557,A -85,B 0,C 180,E1 -22715.11,E2 -22715.11} C_VEL
LIN {X 0,Y 230.56,Z 390.999,A -85,B 0,C 180,E1 -22717.495,E2 -22717.495} C_VEL
LIN {X 0,Y 234.319,Z 400.202,A -85,B 0,C 180,E1 -22719.108,E2 -22719.108} C_VEL
LIN {X 0,Y 233.561,Z 412.418,A -85,B 0,C 180,E1 -22719.461,E2 -22719.461} C_VEL
LIN {X 0,Y 232.677,Z 418.273,A -85,B 0,C 180,E1 -22719.475,E2 -22719.475} C_VEL
LIN {X 0,Y 227.682,Z 437.332,A -85,B 0,C 180,E1 -22718.878,E2 -22718.878} C_VEL
LIN {X 0,Y 226.91,Z 443.177,A -85,B 0,C 180,E1 -22718.925,E2 -22718.925} C_VEL
LIN {X 0,Y 224.164,Z 478.344,A -85,B 0,C 180,E1 -22719.904,E2 -22719.904} C_VEL
LIN {X 0,Y 221.814,Z 494.035,A -85,B 0,C 180,E1 -22720.588,E2 -22720.588} C_VEL
LIN {X 0,Y 218.795,Z 508.51,A -85,B 0,C 180,E1 -22721.513,E2 -22721.513} C_VEL
LIN {X 0,Y 215.13,Z 522.241,A -85,B 0,C 180,E1 -22722.691,E2 -22722.691} C_VEL
LIN {X 0,Y 210.774,Z 535.695,A -85,B 0,C 180,E1 -22724.203,E2 -22724.203} C_VEL
LIN {X 0,Y 205.897,Z 548.899,A -85,B 0,C 180,E1 -22726.143,E2 -22726.143} C_VEL
LIN {X 0,Y 200.199,Z 561.817,A -85,B 0,C 180,E1 -22728.502,E2 -22728.502} C_VEL
LIN {X 0,Y 194.295,Z 573.993,A -85,B 0,C 180,E1 -22731.395,E2 -22731.395} C_VEL
LIN {X 0,Y 188.565,Z 584.832,A -85,B 0,C 180,E1 -22734.712,E2 -22734.712} C_VEL
LIN {X 0,Y 183.644,Z 593.872,A -85,B 0,C 180,E1 -22738.251,E2 -22738.251} C_VEL
LIN {X 0,Y 179.201,Z 601.371,A -85,B 0,C 180,E1 -22741.926,E2 -22741.926} C_VEL
LIN {X 0,Y 175.208,Z 608.377,A -85,B 0,C 180,E1 -22746.352,E2 -22746.352} C_VEL
LIN {X 0,Y 172.251,Z 613.895,A -85,B 0,C 180,E1 -22750.95,E2 -22750.95} C_VEL
LIN {X 0,Y 170.183,Z 618.071,A -85,B 0,C 180,E1 -22755.654,E2 -22755.654} C_VEL
LIN {X 0,Y 169.15,Z 621.009,A -85,B 0,C 180,E1 -22760.434,E2 -22760.434} C_VEL
LIN {X 0,Y 168.798,Z 622.766,A -85,B 0,C 180,E1 -22765.223,E2 -22765.223} C_VEL
LIN {X 0,Y 168.983,Z 623.373,A -85,B 0,C 180,E1 -22770,E2 -22770} C_VEL
LIN {X 0,Y 168.792,Z 622.75,A -85,B 0,C 180,E1 -22774.777,E2 -22774.777} C_VEL
LIN {X 0,Y 169.124,Z 620.971,A -85,B 0,C 180,E1 -22779.568,E2 -22779.568} C_VEL
LIN {X 0,Y 170.174,Z 618.016,A -85,B 0,C 180,E1 -22784.347,E2 -22784.347} C_VEL
LIN {X 0,Y 172.201,Z 613.824,A -85,B 0,C 180,E1 -22789.056,E2 -22789.056} C_VEL
LIN {X 0,Y 175.2,Z 608.282,A -85,B 0,C 180,E1 -22793.649,E2 -22793.649} C_VEL
LIN {X 0,Y 179.215,Z 601.245,A -85,B 0,C 180,E1 -22798.071,E2 -22798.071} C_VEL
LIN {X 0,Y 183.678,Z 593.731,A -85,B 0,C 180,E1 -22801.742,E2 -22801.742} C_VEL
LIN {X 0,Y 188.582,Z 584.669,A -85,B 0,C 180,E1 -22805.284,E2 -22805.284} C_VEL
LIN {X 0,Y 194.309,Z 573.788,A -85,B 0,C 180,E1 -22808.602,E2 -22808.602} C_VEL
LIN {X 0,Y 200.181,Z 561.558,A -85,B 0,C 180,E1 -22811.502,E2 -22811.502} C_VEL
LIN {X 0,Y 205.43,Z 549.723,A -85,B 0,C 180,E1 -22813.681,E2 -22813.681} C_VEL
LIN {X 0,Y 210.242,Z 536.835,A -85,B 0,C 180,E1 -22815.603,E2 -22815.603} C_VEL
LIN {X 0,Y 214.534,Z 523.581,A -85,B 0,C 180,E1 -22817.136,E2 -22817.136} C_VEL
LIN {X 0,Y 218.241,Z 510.21,A -85,B 0,C 180,E1 -22818.304,E2 -22818.304} C_VEL
LIN {X 0,Y 221.4,Z 495.57,A -85,B 0,C 180,E1 -22819.275,E2 -22819.275} C_VEL
LIN {X 0,Y 223.679,Z 480.726,A -85,B 0,C 180,E1 -22819.973,E2 -22819.973} C_VEL
LIN {X 0,Y 225.482,Z 461.044,A -85,B 0,C 180,E1 -22820.55,E2 -22820.55} C_VEL
LIN {X 0,Y 229.554,Z 402.589,A -85,B 0,C 180,E1 -22822.158,E2 -22822.158} C_VEL
LIN {X 0,Y 224.318,Z 389.91,A -85,B 0,C 180,E1 -22824.577,E2 -22824.577} C_VEL
LIN {X 0,Y 219.206,Z 379.178,A -85,B 0,C 180,E1 -22827.11,E2 -22827.11} C_VEL
LIN {X 0,Y 214.408,Z 369.97,A -85,B 0,C 180,E1 -22829.721,E2 -22829.721} C_VEL
LIN {X 0,Y 210.241,Z 362.708,A -85,B 0,C 180,E1 -22832.221,E2 -22832.221} C_VEL
LIN {X 0,Y 207.62,Z 359.026,A -85,B 0,C 180,E1 -22833.893,E2 -22833.893} C_VEL
LIN {X 0,Y 204.866,Z 355.159,A -85,B 0,C 180,E1 -22835.814,E2 -22835.814} C_VEL
LIN {X 0,Y 202.189,Z 351.485,A -85,B 0,C 180,E1 -22837.877,E2 -22837.877} C_VEL
LIN {X 0,Y 198.994,Z 347.677,A -85,B 0,C 180,E1 -22840.631,E2 -22840.631} C_VEL
LIN {X 0,Y 198.001,Z 346.022,A -85,B 0,C 180,E1 -22841.638,E2 -22841.638} C_VEL
LIN {X 0,Y 195.461,Z 343.451,A -85,B 0,C 180,E1 -22844.332,E2 -22844.332} C_VEL
LIN {X 0,Y 193.964,Z 340.708,A -85,B 0,C 180,E1 -22846.378,E2 -22846.378} C_VEL
LIN {X 0,Y 191.481,Z 338.704,A -85,B 0,C 180,E1 -22850.227,E2 -22850.227} C_VEL
LIN {X 0,Y 189.898,Z 335.125,A -85,B 0,C 180,E1 -22854.691,E2 -22854.691} C_VEL
LIN {X 0,Y 189.069,Z 334.684,A -85,B 0,C 180,E1 -22860,E2 -22860} C_VEL
LIN {X 0,Y 190.029,Z 335.371,A -85,B 0,C 180,E1 -22866.237,E2 -22866.237} C_VEL
LIN {X 0,Y 191.259,Z 338.48,A -85,B 0,C 180,E1 -22869.785,E2 -22869.785} C_VEL
LIN {X 0,Y 193.629,Z 340.609,A -85,B 0,C 180,E1 -22873.646,E2 -22873.646} C_VEL
LIN {X 0,Y 194.287,Z 341.277,A -85,B 0,C 180,E1 -22874.534,E2 -22874.534} C_VEL
LIN {X 0,Y 196.26,Z 344.537,A -85,B 0,C 180,E1 -22877.049,E2 -22877.049} C_VEL
LIN {X 0,Y 198.389,Z 346.537,A -85,B 0,C 180,E1 -22879.196,E2 -22879.196} C_VEL
LIN {X 0,Y 200.748,Z 349.993,A -85,B 0,C 180,E1 -22881.403,E2 -22881.403} C_VEL
LIN {X 0,Y 202.308,Z 351.655,A -85,B 0,C 180,E1 -22882.668,E2 -22882.668} C_VEL
LIN {X 0,Y 205.129,Z 355.421,A -85,B 0,C 180,E1 -22884.817,E2 -22884.817} C_VEL
LIN {X 0,Y 209.29,Z 361.36,A -85,B 0,C 180,E1 -22887.635,E2 -22887.635} C_VEL
LIN {X 0,Y 212.824,Z 366.464,A -85,B 0,C 180,E1 -22889.76,E2 -22889.76} C_VEL
LIN {X 0,Y 218.48,Z 375.224,A -85,B 0,C 180,E1 -22892.809,E2 -22892.809} C_VEL
LIN {X 0,Y 225.274,Z 386.969,A -85,B 0,C 180,E1 -22896.052,E2 -22896.052} C_VEL
LIN {X 0,Y 229.993,Z 396.065,A -85,B 0,C 180,E1 -22898.105,E2 -22898.105} C_VEL
LIN {X 0,Y 224.65,Z 469.189,A -85,B 0,C 180,E1 -22900.117,E2 -22900.117} C_VEL
LIN {X 0,Y 222.456,Z 484.595,A -85,B 0,C 180,E1 -22900.78,E2 -22900.78} C_VEL
LIN {X 0,Y 219.632,Z 499.299,A -85,B 0,C 180,E1 -22901.759,E2 -22901.759} C_VEL
LIN {X 0,Y 215.863,Z 514.158,A -85,B 0,C 180,E1 -22903.089,E2 -22903.089} C_VEL
LIN {X 0,Y 211.611,Z 528.177,A -85,B 0,C 180,E1 -22904.775,E2 -22904.775} C_VEL
LIN {X 0,Y 206.506,Z 541.619,A -85,B 0,C 180,E1 -22906.773,E2 -22906.773} C_VEL
LIN {X 0,Y 201.349,Z 553.814,A -85,B 0,C 180,E1 -22909.123,E2 -22909.123} C_VEL
LIN {X 0,Y 195.922,Z 564.93,A -85,B 0,C 180,E1 -22911.774,E2 -22911.774} C_VEL
LIN {X 0,Y 192.486,Z 571.695,A -85,B 0,C 180,E1 -22913.776,E2 -22913.776} C_VEL
LIN {X 0,Y 188.102,Z 579.744,A -85,B 0,C 180,E1 -22916.559,E2 -22916.559} C_VEL
LIN {X 0,Y 183.336,Z 587.992,A -85,B 0,C 180,E1 -22920.111,E2 -22920.111} C_VEL
LIN {X 0,Y 178.65,Z 595.737,A -85,B 0,C 180,E1 -22924.36,E2 -22924.36} C_VEL
LIN {X 0,Y 175.055,Z 601.89,A -85,B 0,C 180,E1 -22928.819,E2 -22928.819} C_VEL
LIN {X 0,Y 172.236,Z 606.638,A -85,B 0,C 180,E1 -22933.404,E2 -22933.404} C_VEL
LIN {X 0,Y 170.492,Z 610.105,A -85,B 0,C 180,E1 -22938.106,E2 -22938.106} C_VEL
LIN {X 0,Y 169.421,Z 612.393,A -85,B 0,C 180,E1 -22942.851,E2 -22942.851} C_VEL
LIN {X 0,Y 169.01,Z 613.555,A -85,B 0,C 180,E1 -22947.617,E2 -22947.617} C_VEL
LIN {X 0,Y 169.027,Z 613.708,A -85,B 0,C 180,E1 -22950,E2 -22950} C_VEL
LIN {X 0,Y 169.146,Z 613.146,A -85,B 0,C 180,E1 -22954.767,E2 -22954.767} C_VEL
LIN {X 0,Y 169.837,Z 611.473,A -85,B 0,C 180,E1 -22959.527,E2 -22959.527} C_VEL
LIN {X 0,Y 171.196,Z 608.646,A -85,B 0,C 180,E1 -22964.259,E2 -22964.259} C_VEL
LIN {X 0,Y 173.525,Z 604.591,A -85,B 0,C 180,E1 -22968.905,E2 -22968.905} C_VEL
LIN {X 0,Y 176.741,Z 599.21,A -85,B 0,C 180,E1 -22973.43,E2 -22973.43} C_VEL
LIN {X 0,Y 180.813,Z 592.349,A -85,B 0,C 180,E1 -22977.802,E2 -22977.802} C_VEL
LIN {X 0,Y 185.887,Z 583.776,A -85,B 0,C 180,E1 -22981.958,E2 -22981.958} C_VEL
LIN {X 0,Y 191.066,Z 574.654,A -85,B 0,C 180,E1 -22985.403,E2 -22985.403} C_VEL
LIN {X 0,Y 194.993,Z 566.984,A -85,B 0,C 180,E1 -22987.785,E2 -22987.785} C_VEL
LIN {X 0,Y 200.302,Z 556.263,A -85,B 0,C 180,E1 -22990.473,E2 -22990.473} C_VEL
LIN {X 0,Y 205.415,Z 544.557,A -85,B 0,C 180,E1 -22992.842,E2 -22992.842} C_VEL
LIN {X 0,Y 210.456,Z 531.761,A -85,B 0,C 180,E1 -22994.864,E2 -22994.864} C_VEL
LIN {X 0,Y 214.945,Z 517.846,A -85,B 0,C 180,E1 -22996.636,E2 -22996.636} C_VEL
LIN {X 0,Y 218.699,Z 503.863,A -85,B 0,C 180,E1 -22997.997,E2 -22997.997} C_VEL
LIN {X 0,Y 221.811,Z 489.196,A -85,B 0,C 180,E1 -22999.066,E2 -22999.066} C_VEL
LIN {X 0,Y 224.161,Z 474.106,A -85,B 0,C 180,E1 -22999.835,E2 -22999.835} C_VEL
LIN {X 0,Y 225.781,Z 456.999,A -85,B 0,C 180,E1 -23000.388,E2 -23000.388} C_VEL
LIN {X 0,Y 230.129,Z 396.076,A -85,B 0,C 180,E1 -23002.033,E2 -23002.033} C_VEL
LIN {X 0,Y 223.902,Z 384.338,A -85,B 0,C 180,E1 -23004.776,E2 -23004.776} C_VEL
LIN {X 0,Y 218.039,Z 374.44,A -85,B 0,C 180,E1 -23007.631,E2 -23007.631} C_VEL
LIN {X 0,Y 212.771,Z 366.323,A -85,B 0,C 180,E1 -23010.504,E2 -23010.504} C_VEL
LIN {X 0,Y 210.051,Z 362.391,A -85,B 0,C 180,E1 -23012.136,E2 -23012.136} C_VEL
LIN {X 0,Y 207.703,Z 359.041,A -85,B 0,C 180,E1 -23013.652,E2 -23013.652} C_VEL
LIN {X 0,Y 204.958,Z 355.234,A -85,B 0,C 180,E1 -23015.577,E2 -23015.577} C_VEL
LIN {X 0,Y 201.619,Z 350.795,A -85,B 0,C 180,E1 -23018.194,E2 -23018.194} C_VEL
LIN {X 0,Y 198.876,Z 347.346,A -85,B 0,C 180,E1 -23020.652,E2 -23020.652} C_VEL
LIN {X 0,Y 198.167,Z 346.14,A -85,B 0,C 180,E1 -23021.386,E2 -23021.386} C_VEL
LIN {X 0,Y 195.522,Z 343.472,A -85,B 0,C 180,E1 -23024.226,E2 -23024.226} C_VEL
LIN {X 0,Y 193.974,Z 340.74,A -85,B 0,C 180,E1 -23026.378,E2 -23026.378} C_VEL
LIN {X 0,Y 191.452,Z 338.628,A -85,B 0,C 180,E1 -23030.491,E2 -23030.491} C_VEL
LIN {X 0,Y 189.958,Z 335.146,A -85,B 0,C 180,E1 -23035.225,E2 -23035.225} C_VEL
LIN {X 0,Y 189.388,Z 334.813,A -85,B 0,C 180,E1 -23040,E2 -23040} C_VEL
LIN {X 0,Y 190.042,Z 335.26,A -85,B 0,C 180,E1 -23044.773,E2 -23044.773} C_VEL
LIN {X 0,Y 192.033,Z 339.347,A -85,B 0,C 180,E1 -23050.299,E2 -23050.299} C_VEL
LIN {X 0,Y 194.217,Z 341.026,A -85,B 0,C 180,E1 -23053.604,E2 -23053.604} C_VEL
LIN {X 0,Y 196.22,Z 344.403,A -85,B 0,C 180,E1 -23056.249,E2 -23056.249} C_VEL
LIN {X 0,Y 198.423,Z 346.545,A -85,B 0,C 180,E1 -23058.522,E2 -23058.522} C_VEL
LIN {X 0,Y 201.061,Z 350.284,A -85,B 0,C 180,E1 -23060.995,E2 -23060.995} C_VEL
LIN {X 0,Y 202.433,Z 351.802,A -85,B 0,C 180,E1 -23062.115,E2 -23062.115} C_VEL
LIN {X 0,Y 206.084,Z 356.808,A -85,B 0,C 180,E1 -23064.88,E2 -23064.88} C_VEL
LIN {X 0,Y 209.639,Z 361.759,A -85,B 0,C 180,E1 -23067.246,E2 -23067.246} C_VEL
LIN {X 0,Y 211.778,Z 365.159,A -85,B 0,C 180,E1 -23068.577,E2 -23068.577} C_VEL
LIN {X 0,Y 216.66,Z 374.011,A -85,B 0,C 180,E1 -23071.401,E2 -23071.401} C_VEL
LIN {X 0,Y 221.91,Z 384.495,A -85,B 0,C 180,E1 -23074.136,E2 -23074.136} C_VEL
LIN {X 0,Y 227.177,Z 396.353,A -85,B 0,C 180,E1 -23076.653,E2 -23076.653} C_VEL
LIN {X 0,Y 229.705,Z 402.698,A -85,B 0,C 180,E1 -23077.804,E2 -23077.804} C_VEL
LIN {X 0,Y 226.91,Z 443.177,A -85,B 0,C 180,E1 -23078.925,E2 -23078.925} C_VEL
LIN {X 0,Y 226.137,Z 449.023,A -85,B 0,C 180,E1 -23078.968,E2 -23078.968} C_VEL
LIN {X 0,Y 221.094,Z 468.059,A -85,B 0,C 180,E1 -23078.32,E2 -23078.32} C_VEL
LIN {X 0,Y 220.141,Z 473.899,A -85,B 0,C 180,E1 -23078.353,E2 -23078.353} C_VEL
LIN {X 0,Y 218.013,Z 489.638,A -85,B 0,C 180,E1 -23078.961,E2 -23078.961} C_VEL
LIN {X 0,Y 215.068,Z 504.522,A -85,B 0,C 180,E1 -23079.833,E2 -23079.833} C_VEL
LIN {X 0,Y 211.502,Z 518.069,A -85,B 0,C 180,E1 -23080.893,E2 -23080.893} C_VEL
LIN {X 0,Y 206.978,Z 532.328,A -85,B 0,C 180,E1 -23082.396,E2 -23082.396} C_VEL
LIN {X 0,Y 202.144,Z 545.323,A -85,B 0,C 180,E1 -23084.188,E2 -23084.188} C_VEL
LIN {X 0,Y 196.975,Z 557.327,A -85,B 0,C 180,E1 -23086.269,E2 -23086.269} C_VEL
LIN {X 0,Y 191.535,Z 568.448,A -85,B 0,C 180,E1 -23088.665,E2 -23088.665} C_VEL
LIN {X 0,Y 186.097,Z 578.695,A -85,B 0,C 180,E1 -23091.456,E2 -23091.456} C_VEL
LIN {X 0,Y 180.502,Z 588.513,A -85,B 0,C 180,E1 -23094.85,E2 -23094.85} C_VEL
LIN {X 0,Y 175.535,Z 597.043,A -85,B 0,C 180,E1 -23098.636,E2 -23098.636} C_VEL
LIN {X 0,Y 171.747,Z 603.044,A -85,B 0,C 180,E1 -23101.928,E2 -23101.928} C_VEL
LIN {X 0,Y 167.744,Z 609.667,A -85,B 0,C 180,E1 -23106.546,E2 -23106.546} C_VEL
LIN {X 0,Y 164.831,Z 614.858,A -85,B 0,C 180,E1 -23111.351,E2 -23111.351} C_VEL
LIN {X 0,Y 163.256,Z 617.867,A -85,B 0,C 180,E1 -23115.032,E2 -23115.032} C_VEL
LIN {X 0,Y 162.11,Z 620.806,A -85,B 0,C 180,E1 -23120.014,E2 -23120.014} C_VEL
LIN {X 0,Y 161.711,Z 622.563,A -85,B 0,C 180,E1 -23125.014,E2 -23125.014} C_VEL
LIN {X 0,Y 161.894,Z 623.17,A -85,B 0,C 180,E1 -23130,E2 -23130} C_VEL
LIN {X 0,Y 161.705,Z 622.546,A -85,B 0,C 180,E1 -23134.986,E2 -23134.986} C_VEL
LIN {X 0,Y 162.088,Z 620.766,A -85,B 0,C 180,E1 -23139.987,E2 -23139.987} C_VEL
LIN {X 0,Y 163.246,Z 617.811,A -85,B 0,C 180,E1 -23144.969,E2 -23144.969} C_VEL
LIN {X 0,Y 165.442,Z 613.618,A -85,B 0,C 180,E1 -23149.867,E2 -23149.867} C_VEL
LIN {X 0,Y 168.645,Z 608.076,A -85,B 0,C 180,E1 -23154.628,E2 -23154.628} C_VEL
LIN {X 0,Y 172.922,Z 601.038,A -85,B 0,C 180,E1 -23159.189,E2 -23159.189} C_VEL
LIN {X 0,Y 177.595,Z 593.523,A -85,B 0,C 180,E1 -23162.964,E2 -23162.964} C_VEL
LIN {X 0,Y 182.775,Z 584.462,A -85,B 0,C 180,E1 -23166.583,E2 -23166.583} C_VEL
LIN {X 0,Y 188.785,Z 573.581,A -85,B 0,C 180,E1 -23169.953,E2 -23169.953} C_VEL
LIN {X 0,Y 194.393,Z 562.383,A -85,B 0,C 180,E1 -23172.677,E2 -23172.677} C_VEL
LIN {X 0,Y 200.262,Z 549.705,A -85,B 0,C 180,E1 -23175.055,E2 -23175.055} C_VEL
LIN {X 0,Y 204.765,Z 538.057,A -85,B 0,C 180,E1 -23176.83,E2 -23176.83} C_VEL
LIN {X 0,Y 209.188,Z 525.141,A -85,B 0,C 180,E1 -23178.374,E2 -23178.374} C_VEL
LIN {X 0,Y 213.28,Z 511.13,A -85,B 0,C 180,E1 -23179.64,E2 -23179.64} C_VEL
LIN {X 0,Y 216.687,Z 496.121,A -85,B 0,C 180,E1 -23180.653,E2 -23180.653} C_VEL
LIN {X 0,Y 219.085,Z 481.181,A -85,B 0,C 180,E1 -23181.372,E2 -23181.372} C_VEL
LIN {X 0,Y 221.005,Z 461.326,A -85,B 0,C 180,E1 -23181.956,E2 -23181.956} C_VEL
LIN {X 0,Y 225.097,Z 405.562,A -85,B 0,C 180,E1 -23183.476,E2 -23183.476} C_VEL
LIN {X 0,Y 221.823,Z 397.097,A -85,B 0,C 180,E1 -23185.087,E2 -23185.087} C_VEL
LIN {X 0,Y 217.245,Z 386.731,A -85,B 0,C 180,E1 -23187.457,E2 -23187.457} C_VEL
LIN {X 0,Y 212.142,Z 376.482,A -85,B 0,C 180,E1 -23190.34,E2 -23190.34} C_VEL
LIN {X 0,Y 208.114,Z 369.06,A -85,B 0,C 180,E1 -23192.872,E2 -23192.872} C_VEL
LIN {X 0,Y 205.113,Z 364.802,A -85,B 0,C 180,E1 -23194.878,E2 -23194.878} C_VEL
LIN {X 0,Y 202.698,Z 361.317,A -85,B 0,C 180,E1 -23196.661,E2 -23196.661} C_VEL
LIN {X 0,Y 199.811,Z 357.338,A -85,B 0,C 180,E1 -23199.022,E2 -23199.022} C_VEL
LIN {X 0,Y 196.924,Z 353.469,A -85,B 0,C 180,E1 -23201.736,E2 -23201.736} C_VEL
LIN {X 0,Y 196.248,Z 352.535,A -85,B 0,C 180,E1 -23202.445,E2 -23202.445} C_VEL
LIN {X 0,Y 193.77,Z 349.668,A -85,B 0,C 180,E1 -23205.293,E2 -23205.293} C_VEL
LIN {X 0,Y 192.724,Z 347.628,A -85,B 0,C 180,E1 -23206.826,E2 -23206.826} C_VEL
LIN {X 0,Y 190.175,Z 345.271,A -85,B 0,C 180,E1 -23211.098,E2 -23211.098} C_VEL
LIN {X 0,Y 188.956,Z 342.156,A -85,B 0,C 180,E1 -23214.932,E2 -23214.932} C_VEL
LIN {X 0,Y 188.206,Z 341.714,A -85,B 0,C 180,E1 -23220,E2 -23220} C_VEL
LIN {X 0,Y 189.044,Z 342.345,A -85,B 0,C 180,E1 -23225.868,E2 -23225.868} C_VEL
LIN {X 0,Y 190.389,Z 345.665,A -85,B 0,C 180,E1 -23229.83,E2 -23229.83} C_VEL
LIN {X 0,Y 192.95,Z 348.036,A -85,B 0,C 180,E1 -23233.964,E2 -23233.964} C_VEL
LIN {X 0,Y 194.955,Z 351.369,A -85,B 0,C 180,E1 -23236.627,E2 -23236.627} C_VEL
LIN {X 0,Y 196.838,Z 353.234,A -85,B 0,C 180,E1 -23238.609,E2 -23238.609} C_VEL
LIN {X 0,Y 199.368,Z 356.847,A -85,B 0,C 180,E1 -23241.047,E2 -23241.047} C_VEL
LIN {X 0,Y 200.528,Z 358.227,A -85,B 0,C 180,E1 -23242.032,E2 -23242.032} C_VEL
LIN {X 0,Y 203.916,Z 363.024,A -85,B 0,C 180,E1 -23244.702,E2 -23244.702} C_VEL
LIN {X 0,Y 207.45,Z 368.112,A -85,B 0,C 180,E1 -23247.148,E2 -23247.148} C_VEL
LIN {X 0,Y 212.022,Z 375.015,A -85,B 0,C 180,E1 -23249.953,E2 -23249.953} C_VEL
LIN {X 0,Y 217.617,Z 384.279,A -85,B 0,C 180,E1 -23252.996,E2 -23252.996} C_VEL
LIN {X 0,Y 224.027,Z 396.099,A -85,B 0,C 180,E1 -23256.1,E2 -23256.1} C_VEL
LIN {X 0,Y 225.514,Z 399.033,A -85,B 0,C 180,E1 -23256.773,E2 -23256.773} C_VEL
LIN {X 0,Y 220.176,Z 469.215,A -85,B 0,C 180,E1 -23258.7,E2 -23258.7} C_VEL
LIN {X 0,Y 217.887,Z 484.808,A -85,B 0,C 180,E1 -23259.367,E2 -23259.367} C_VEL
LIN {X 0,Y 214.709,Z 500.663,A -85,B 0,C 180,E1 -23260.446,E2 -23260.446} C_VEL
LIN {X 0,Y 210.939,Z 514.864,A -85,B 0,C 180,E1 -23261.739,E2 -23261.739} C_VEL
LIN {X 0,Y 206.66,Z 528.385,A -85,B 0,C 180,E1 -23263.374,E2 -23263.374} C_VEL
LIN {X 0,Y 201.391,Z 541.826,A -85,B 0,C 180,E1 -23265.389,E2 -23265.389} C_VEL
LIN {X 0,Y 196.024,Z 554.021,A -85,B 0,C 180,E1 -23267.762,E2 -23267.762} C_VEL
LIN {X 0,Y 190.375,Z 565.137,A -85,B 0,C 180,E1 -23270.447,E2 -23270.447} C_VEL
LIN {X 0,Y 186.175,Z 572.997,A -85,B 0,C 180,E1 -23272.845,E2 -23272.845} C_VEL
LIN {X 0,Y 181.442,Z 581.211,A -85,B 0,C 180,E1 -23275.831,E2 -23275.831} C_VEL
LIN {X 0,Y 176.536,Z 589.283,A -85,B 0,C 180,E1 -23279.498,E2 -23279.498} C_VEL
LIN {X 0,Y 171.572,Z 597.017,A -85,B 0,C 180,E1 -23284.045,E2 -23284.045} C_VEL
LIN {X 0,Y 167.592,Z 603.408,A -85,B 0,C 180,E1 -23289.118,E2 -23289.118} C_VEL
LIN {X 0,Y 165.409,Z 606.843,A -85,B 0,C 180,E1 -23292.698,E2 -23292.698} C_VEL
LIN {X 0,Y 163.513,Z 610.31,A -85,B 0,C 180,E1 -23297.59,E2 -23297.59} C_VEL
LIN {X 0,Y 162.376,Z 612.596,A -85,B 0,C 180,E1 -23302.54,E2 -23302.54} C_VEL
LIN {X 0,Y 161.926,Z 613.757,A -85,B 0,C 180,E1 -23307.513,E2 -23307.513} C_VEL
LIN {X 0,Y 161.939,Z 613.91,A -85,B 0,C 180,E1 -23310,E2 -23310} C_VEL
LIN {X 0,Y 162.067,Z 613.349,A -85,B 0,C 180,E1 -23314.975,E2 -23314.975} C_VEL
LIN {X 0,Y 162.825,Z 611.676,A -85,B 0,C 180,E1 -23319.942,E2 -23319.942} C_VEL
LIN {X 0,Y 164.29,Z 608.85,A -85,B 0,C 180,E1 -23324.872,E2 -23324.872} C_VEL
LIN {X 0,Y 166.809,Z 604.794,A -85,B 0,C 180,E1 -23329.697,E2 -23329.697} C_VEL
LIN {X 0,Y 170.221,Z 599.413,A -85,B 0,C 180,E1 -23334.385,E2 -23334.385} C_VEL
LIN {X 0,Y 174.543,Z 592.551,A -85,B 0,C 180,E1 -23338.893,E2 -23338.893} C_VEL
LIN {X 0,Y 179.858,Z 583.978,A -85,B 0,C 180,E1 -23343.164,E2 -23343.164} C_VEL
LIN {X 0,Y 185.279,Z 574.856,A -85,B 0,C 180,E1 -23346.685,E2 -23346.685} C_VEL
LIN {X 0,Y 189.42,Z 567.185,A -85,B 0,C 180,E1 -23349.104,E2 -23349.104} C_VEL
LIN {X 0,Y 194.949,Z 556.463,A -85,B 0,C 180,E1 -23351.829,E2 -23351.829} C_VEL
LIN {X 0,Y 200.267,Z 544.756,A -85,B 0,C 180,E1 -23354.223,E2 -23354.223} C_VEL
LIN {X 0,Y 205.478,Z 531.996,A -85,B 0,C 180,E1 -23356.254,E2 -23356.254} C_VEL
LIN {X 0,Y 210.201,Z 517.842,A -85,B 0,C 180,E1 -23358.063,E2 -23358.063} C_VEL
LIN {X 0,Y 214.283,Z 502.932,A -85,B 0,C 180,E1 -23359.506,E2 -23359.506} C_VEL
LIN {X 0,Y 217.53,Z 487.867,A -85,B 0,C 180,E1 -23360.565,E2 -23360.565} C_VEL
LIN {X 0,Y 219.884,Z 472.705,A -85,B 0,C 180,E1 -23361.302,E2 -23361.302} C_VEL
LIN {X 0,Y 221.734,Z 452.192,A -85,B 0,C 180,E1 -23361.925,E2 -23361.925} C_VEL
LIN {X 0,Y 225.631,Z 399.094,A -85,B 0,C 180,E1 -23363.373,E2 -23363.373} C_VEL
LIN {X 0,Y 219.918,Z 388.233,A -85,B 0,C 180,E1 -23366.059,E2 -23366.059} C_VEL
LIN {X 0,Y 215.001,Z 379.78,A -85,B 0,C 180,E1 -23368.602,E2 -23368.602} C_VEL
LIN {X 0,Y 210.413,Z 372.448,A -85,B 0,C 180,E1 -23371.237,E2 -23371.237} C_VEL
LIN {X 0,Y 205.881,Z 365.688,A -85,B 0,C 180,E1 -23374.174,E2 -23374.174} C_VEL
LIN {X 0,Y 202.707,Z 361.201,A -85,B 0,C 180,E1 -23376.502,E2 -23376.502} C_VEL
LIN {X 0,Y 199.839,Z 357.3,A -85,B 0,C 180,E1 -23378.87,E2 -23378.87} C_VEL
LIN {X 0,Y 197.15,Z 353.686,A -85,B 0,C 180,E1 -23381.421,E2 -23381.421} C_VEL
LIN {X 0,Y 196.33,Z 352.585,A -85,B 0,C 180,E1 -23382.285,E2 -23382.285} C_VEL
LIN {X 0,Y 193.941,Z 349.849,A -85,B 0,C 180,E1 -23385.061,E2 -23385.061} C_VEL
LIN {X 0,Y 192.75,Z 347.628,A -85,B 0,C 180,E1 -23386.827,E2 -23386.827} C_VEL
LIN {X 0,Y 190.347,Z 345.458,A -85,B 0,C 180,E1 -23390.972,E2 -23390.972} C_VEL
LIN {X 0,Y 189.085,Z 342.191,A -85,B 0,C 180,E1 -23395.241,E2 -23395.241} C_VEL
LIN {X 0,Y 188.523,Z 341.861,A -85,B 0,C 180,E1 -23400,E2 -23400} C_VEL
LIN {X 0,Y 189.104,Z 342.321,A -85,B 0,C 180,E1 -23404.529,E2 -23404.529} C_VEL
LIN {X 0,Y 191.018,Z 346.331,A -85,B 0,C 180,E1 -23410.065,E2 -23410.065} C_VEL
LIN {X 0,Y 192.98,Z 347.929,A -85,B 0,C 180,E1 -23413.156,E2 -23413.156} C_VEL
LIN {X 0,Y 195.029,Z 351.369,A -85,B 0,C 180,E1 -23415.948,E2 -23415.948} C_VEL
LIN {X 0,Y 196.938,Z 353.345,A -85,B 0,C 180,E1 -23417.996,E2 -23417.996} C_VEL
LIN {X 0,Y 199.789,Z 357.249,A -85,B 0,C 180,E1 -23420.73,E2 -23420.73} C_VEL
LIN {X 0,Y 201.109,Z 359.062,A -85,B 0,C 180,E1 -23421.863,E2 -23421.863} C_VEL
LIN {X 0,Y 204.133,Z 363.263,A -85,B 0,C 180,E1 -23424.226,E2 -23424.226} C_VEL
LIN {X 0,Y 207.372,Z 367.871,A -85,B 0,C 180,E1 -23426.479,E2 -23426.479} C_VEL
LIN {X 0,Y 209.075,Z 370.667,A -85,B 0,C 180,E1 -23427.597,E2 -23427.597} C_VEL
LIN {X 0,Y 213.669,Z 379.262,A -85,B 0,C 180,E1 -23430.413,E2 -23430.413} C_VEL
LIN {X 0,Y 218.681,Z 389.65,A -85,B 0,C 180,E1 -23433.179,E2 -23433.179} C_VEL
LIN {X 0,Y 223.432,Z 400.681,A -85,B 0,C 180,E1 -23435.585,E2 -23435.585} C_VEL
LIN {X 0,Y 225.186,Z 405.218,A -85,B 0,C 180,E1 -23436.438,E2 -23436.438} C_VEL
LIN {X 0,Y 222.927,Z 437.433,A -85,B 0,C 180,E1 -23437.352,E2 -23437.352} C_VEL
LIN {X 0,Y 220.141,Z 473.899,A -85,B 0,C 180,E1 -23438.353,E2 -23438.353} C_VEL
LIN {X 0,Y 219.079,Z 479.71,A -85,B 0,C 180,E1 -23438.404,E2 -23438.404} C_VEL
LIN {X 0,Y 215.89,Z 489.075,A -85,B 0,C 180,E1 -23438.203,E2 -23438.203} C_VEL
LIN {X 0,Y 212.331,Z 498.373,A -85,B 0,C 180,E1 -23438.099,E2 -23438.099} C_VEL
LIN {X 0,Y 210.688,Z 503.913,A -85,B 0,C 180,E1 -23438.322,E2 -23438.322} C_VEL
LIN {X 0,Y 206.926,Z 517.872,A -85,B 0,C 180,E1 -23439.407,E2 -23439.407} C_VEL
LIN {X 0,Y 202.26,Z 532.129,A -85,B 0,C 180,E1 -23440.911,E2 -23440.911} C_VEL
LIN {X 0,Y 197.213,Z 545.122,A -85,B 0,C 180,E1 -23442.695,E2 -23442.695} C_VEL
LIN {X 0,Y 191.874,Z 557.126,A -85,B 0,C 180,E1 -23444.793,E2 -23444.793} C_VEL
LIN {X 0,Y 186.226,Z 568.247,A -85,B 0,C 180,E1 -23447.212,E2 -23447.212} C_VEL
LIN {X 0,Y 180.559,Z 578.493,A -85,B 0,C 180,E1 -23450.042,E2 -23450.042} C_VEL
LIN {X 0,Y 174.328,Z 588.907,A -85,B 0,C 180,E1 -23453.735,E2 -23453.735} C_VEL
LIN {X 0,Y 168.77,Z 597.921,A -85,B 0,C 180,E1 -23457.932,E2 -23457.932} C_VEL
LIN {X 0,Y 164.287,Z 604.665,A -85,B 0,C 180,E1 -23461.93,E2 -23461.93} C_VEL
LIN {X 0,Y 160.285,Z 610.902,A -85,B 0,C 180,E1 -23466.758,E2 -23466.758} C_VEL
LIN {X 0,Y 157.459,Z 615.736,A -85,B 0,C 180,E1 -23471.794,E2 -23471.794} C_VEL
LIN {X 0,Y 155.602,Z 619.283,A -85,B 0,C 180,E1 -23476.949,E2 -23476.949} C_VEL
LIN {X 0,Y 154.762,Z 621.625,A -85,B 0,C 180,E1 -23482.17,E2 -23482.17} C_VEL
LIN {X 0,Y 154.662,Z 622.808,A -85,B 0,C 180,E1 -23487.396,E2 -23487.396} C_VEL
LIN {X 0,Y 154.793,Z 622.967,A -85,B 0,C 180,E1 -23490,E2 -23490} C_VEL
LIN {X 0,Y 154.62,Z 622.343,A -85,B 0,C 180,E1 -23495.216,E2 -23495.216} C_VEL
LIN {X 0,Y 155.041,Z 620.561,A -85,B 0,C 180,E1 -23500.446,E2 -23500.446} C_VEL
LIN {X 0,Y 156.346,Z 617.606,A -85,B 0,C 180,E1 -23505.646,E2 -23505.646} C_VEL
LIN {X 0,Y 158.69,Z 613.411,A -85,B 0,C 180,E1 -23510.75,E2 -23510.75} C_VEL
LIN {X 0,Y 162.17,Z 607.87,A -85,B 0,C 180,E1 -23515.681,E2 -23515.681} C_VEL
LIN {X 0,Y 166.709,Z 600.832,A -85,B 0,C 180,E1 -23520.389,E2 -23520.389} C_VEL
LIN {X 0,Y 171.602,Z 593.316,A -85,B 0,C 180,E1 -23524.272,E2 -23524.272} C_VEL
LIN {X 0,Y 177.062,Z 584.254,A -85,B 0,C 180,E1 -23527.967,E2 -23527.967} C_VEL
LIN {X 0,Y 183.351,Z 573.374,A -85,B 0,C 180,E1 -23531.391,E2 -23531.391} C_VEL
LIN {X 0,Y 189.219,Z 562.176,A -85,B 0,C 180,E1 -23534.139,E2 -23534.139} C_VEL
LIN {X 0,Y 195.185,Z 549.723,A -85,B 0,C 180,E1 -23536.497,E2 -23536.497} C_VEL
LIN {X 0,Y 199.964,Z 537.85,A -85,B 0,C 180,E1 -23538.317,E2 -23538.317} C_VEL
LIN {X 0,Y 204.529,Z 524.932,A -85,B 0,C 180,E1 -23539.865,E2 -23539.865} C_VEL
LIN {X 0,Y 208.757,Z 510.92,A -85,B 0,C 180,E1 -23541.124,E2 -23541.124} C_VEL
LIN {X 0,Y 212.109,Z 496.672,A -85,B 0,C 180,E1 -23542.09,E2 -23542.09} C_VEL
LIN {X 0,Y 214.633,Z 481.659,A -85,B 0,C 180,E1 -23542.825,E2 -23542.825} C_VEL
LIN {X 0,Y 216.501,Z 463.459,A -85,B 0,C 180,E1 -23543.378,E2 -23543.378} C_VEL
LIN {X 0,Y 220.73,Z 407.887,A -85,B 0,C 180,E1 -23544.893,E2 -23544.893} C_VEL
LIN {X 0,Y 215.946,Z 395.988,A -85,B 0,C 180,E1 -23547.435,E2 -23547.435} C_VEL
LIN {X 0,Y 210.989,Z 385.245,A -85,B 0,C 180,E1 -23550.299,E2 -23550.299} C_VEL
LIN {X 0,Y 206.979,Z 377.415,A -85,B 0,C 180,E1 -23552.861,E2 -23552.861} C_VEL
LIN {X 0,Y 205.17,Z 374.188,A -85,B 0,C 180,E1 -23554.104,E2 -23554.104} C_VEL
LIN {X 0,Y 201.094,Z 368.093,A -85,B 0,C 180,E1 -23557.12,E2 -23557.12} C_VEL
LIN {X 0,Y 198.001,Z 363.765,A -85,B 0,C 180,E1 -23559.753,E2 -23559.753} C_VEL
LIN {X 0,Y 195.214,Z 359.793,A -85,B 0,C 180,E1 -23562.535,E2 -23562.535} C_VEL
LIN {X 0,Y 192.152,Z 355.895,A -85,B 0,C 180,E1 -23566.247,E2 -23566.247} C_VEL
LIN {X 0,Y 191.316,Z 354.42,A -85,B 0,C 180,E1 -23567.537,E2 -23567.537} C_VEL
LIN {X 0,Y 188.97,Z 351.889,A -85,B 0,C 180,E1 -23571.849,E2 -23571.849} C_VEL
LIN {X 0,Y 187.979,Z 349.18,A -85,B 0,C 180,E1 -23575.309,E2 -23575.309} C_VEL
LIN {X 0,Y 187.344,Z 348.738,A -85,B 0,C 180,E1 -23580,E2 -23580} C_VEL
LIN {X 0,Y 188.089,Z 349.468,A -85,B 0,C 180,E1 -23585.629,E2 -23585.629} C_VEL
LIN {X 0,Y 189.716,Z 353.092,A -85,B 0,C 180,E1 -23590.27,E2 -23590.27} C_VEL
LIN {X 0,Y 191.717,Z 354.93,A -85,B 0,C 180,E1 -23593.515,E2 -23593.515} C_VEL
LIN {X 0,Y 193.767,Z 358.321,A -85,B 0,C 180,E1 -23596.326,E2 -23596.326} C_VEL
LIN {X 0,Y 195.336,Z 359.968,A -85,B 0,C 180,E1 -23598.045,E2 -23598.045} C_VEL
LIN {X 0,Y 197.962,Z 363.712,A -85,B 0,C 180,E1 -23600.659,E2 -23600.659} C_VEL
LIN {X 0,Y 201.65,Z 368.894,A -85,B 0,C 180,E1 -23603.765,E2 -23603.765} C_VEL
LIN {X 0,Y 205.707,Z 375.017,A -85,B 0,C 180,E1 -23606.711,E2 -23606.711} C_VEL
LIN {X 0,Y 210.158,Z 382.051,A -85,B 0,C 180,E1 -23609.535,E2 -23609.535} C_VEL
LIN {X 0,Y 215.385,Z 391.098,A -85,B 0,C 180,E1 -23612.482,E2 -23612.482} C_VEL
LIN {X 0,Y 221.119,Z 402.079,A -85,B 0,C 180,E1 -23615.376,E2 -23615.376} C_VEL
LIN {X 0,Y 215.818,Z 469.387,A -85,B 0,C 180,E1 -23617.229,E2 -23617.229} C_VEL
LIN {X 0,Y 213.466,Z 485.021,A -85,B 0,C 180,E1 -23617.898,E2 -23617.898} C_VEL
LIN {X 0,Y 210.455,Z 499.72,A -85,B 0,C 180,E1 -23618.878,E2 -23618.878} C_VEL
LIN {X 0,Y 206.514,Z 514.298,A -85,B 0,C 180,E1 -23620.183,E2 -23620.183} C_VEL
LIN {X 0,Y 201.849,Z 528.593,A -85,B 0,C 180,E1 -23621.908,E2 -23621.908} C_VEL
LIN {X 0,Y 196.388,Z 542.034,A -85,B 0,C 180,E1 -23623.931,E2 -23623.931} C_VEL
LIN {X 0,Y 190.816,Z 554.228,A -85,B 0,C 180,E1 -23626.325,E2 -23626.325} C_VEL
LIN {X 0,Y 184.931,Z 565.344,A -85,B 0,C 180,E1 -23629.04,E2 -23629.04} C_VEL
LIN {X 0,Y 180.504,Z 573.205,A -85,B 0,C 180,E1 -23631.468,E2 -23631.468} C_VEL
LIN {X 0,Y 176.41,Z 580.155,A -85,B 0,C 180,E1 -23634.012,E2 -23634.012} C_VEL
LIN {X 0,Y 171.127,Z 588.404,A -85,B 0,C 180,E1 -23637.732,E2 -23637.732} C_VEL
LIN {X 0,Y 165.901,Z 596.148,A -85,B 0,C 180,E1 -23642.227,E2 -23642.227} C_VEL
LIN {X 0,Y 161.797,Z 602.302,A -85,B 0,C 180,E1 -23646.988,E2 -23646.988} C_VEL
LIN {X 0,Y 158.608,Z 607.048,A -85,B 0,C 180,E1 -23651.931,E2 -23651.931} C_VEL
LIN {X 0,Y 156.56,Z 610.514,A -85,B 0,C 180,E1 -23657.03,E2 -23657.03} C_VEL
LIN {X 0,Y 155.328,Z 612.8,A -85,B 0,C 180,E1 -23662.199,E2 -23662.199} C_VEL
LIN {X 0,Y 154.845,Z 613.96,A -85,B 0,C 180,E1 -23667.399,E2 -23667.399} C_VEL
LIN {X 0,Y 154.853,Z 614.113,A -85,B 0,C 180,E1 -23670,E2 -23670} C_VEL
LIN {X 0,Y 155.005,Z 613.552,A -85,B 0,C 180,E1 -23675.203,E2 -23675.203} C_VEL
LIN {X 0,Y 155.815,Z 611.879,A -85,B 0,C 180,E1 -23680.394,E2 -23680.394} C_VEL
LIN {X 0,Y 157.414,Z 609.053,A -85,B 0,C 180,E1 -23685.538,E2 -23685.538} C_VEL
LIN {X 0,Y 160.096,Z 604.997,A -85,B 0,C 180,E1 -23690.559,E2 -23690.559} C_VEL
LIN {X 0,Y 163.747,Z 599.615,A -85,B 0,C 180,E1 -23695.416,E2 -23695.416} C_VEL
LIN {X 0,Y 168.322,Z 592.754,A -85,B 0,C 180,E1 -23700.068,E2 -23700.068} C_VEL
LIN {X 0,Y 173.923,Z 584.181,A -85,B 0,C 180,E1 -23704.451,E2 -23704.451} C_VEL
LIN {X 0,Y 178.81,Z 576.466,A -85,B 0,C 180,E1 -23707.532,E2 -23707.532} C_VEL
LIN {X 0,Y 183.045,Z 568.957,A -85,B 0,C 180,E1 -23710.044,E2 -23710.044} C_VEL
LIN {X 0,Y 188.713,Z 558.606,A -85,B 0,C 180,E1 -23712.816,E2 -23712.816} C_VEL
LIN {X 0,Y 194.197,Z 547.293,A -85,B 0,C 180,E1 -23715.252,E2 -23715.252} C_VEL
LIN {X 0,Y 199.528,Z 534.991,A -85,B 0,C 180,E1 -23717.329,E2 -23717.329} C_VEL
LIN {X 0,Y 204.409,Z 521.536,A -85,B 0,C 180,E1 -23719.146,E2 -23719.146} C_VEL
LIN {X 0,Y 208.631,Z 507.582,A -85,B 0,C 180,E1 -23720.593,E2 -23720.593} C_VEL
LIN {X 0,Y 212.077,Z 493.238,A -85,B 0,C 180,E1 -23721.716,E2 -23721.716} C_VEL
LIN {X 0,Y 214.875,Z 477.695,A -85,B 0,C 180,E1 -23722.581,E2 -23722.581} C_VEL
LIN {X 0,Y 216.617,Z 462.831,A -85,B 0,C 180,E1 -23723.108,E2 -23723.108} C_VEL
LIN {X 0,Y 221.23,Z 402.109,A -85,B 0,C 180,E1 -23724.778,E2 -23724.778} C_VEL
LIN {X 0,Y 215.343,Z 390.85,A -85,B 0,C 180,E1 -23727.764,E2 -23727.764} C_VEL
LIN {X 0,Y 210.1,Z 381.776,A -85,B 0,C 180,E1 -23730.745,E2 -23730.745} C_VEL
LIN {X 0,Y 205.537,Z 374.615,A -85,B 0,C 180,E1 -23733.673,E2 -23733.673} C_VEL
LIN {X 0,Y 201.235,Z 368.132,A -85,B 0,C 180,E1 -23736.865,E2 -23736.865} C_VEL
LIN {X 0,Y 198.156,Z 363.868,A -85,B 0,C 180,E1 -23739.498,E2 -23739.498} C_VEL
LIN {X 0,Y 195.403,Z 359.943,A -85,B 0,C 180,E1 -23742.266,E2 -23742.266} C_VEL
LIN {X 0,Y 192.459,Z 356.294,A -85,B 0,C 180,E1 -23745.831,E2 -23745.831} C_VEL
LIN {X 0,Y 191.536,Z 354.529,A -85,B 0,C 180,E1 -23747.281,E2 -23747.281} C_VEL
LIN {X 0,Y 189.257,Z 352.274,A -85,B 0,C 180,E1 -23751.457,E2 -23751.457} C_VEL
LIN {X 0,Y 188.103,Z 349.213,A -85,B 0,C 180,E1 -23755.714,E2 -23755.714} C_VEL
LIN {X 0,Y 187.794,Z 349.046,A -85,B 0,C 180,E1 -23762.144,E2 -23762.144} C_VEL
LIN {X 0,Y 188.171,Z 349.37,A -85,B 0,C 180,E1 -23764.284,E2 -23764.284} C_VEL
LIN {X 0,Y 189.968,Z 353.254,A -85,B 0,C 180,E1 -23769.75,E2 -23769.75} C_VEL
LIN {X 0,Y 191.752,Z 354.863,A -85,B 0,C 180,E1 -23772.703,E2 -23772.703} C_VEL
LIN {X 0,Y 194.057,Z 358.571,A -85,B 0,C 180,E1 -23775.895,E2 -23775.895} C_VEL
LIN {X 0,Y 195.436,Z 360.058,A -85,B 0,C 180,E1 -23777.421,E2 -23777.421} C_VEL
LIN {X 0,Y 198.243,Z 363.951,A -85,B 0,C 180,E1 -23780.221,E2 -23780.221} C_VEL
LIN {X 0,Y 202.229,Z 369.716,A -85,B 0,C 180,E1 -23783.571,E2 -23783.571} C_VEL
LIN {X 0,Y 206.057,Z 375.359,A -85,B 0,C 180,E1 -23786.32,E2 -23786.32} C_VEL
LIN {X 0,Y 210.928,Z 384.932,A -85,B 0,C 180,E1 -23789.513,E2 -23789.513} C_VEL
LIN {X 0,Y 215.902,Z 395.692,A -85,B 0,C 180,E1 -23792.408,E2 -23792.408} C_VEL
LIN {X 0,Y 220.215,Z 406.16,A -85,B 0,C 180,E1 -23794.713,E2 -23794.713} C_VEL
LIN {X 0,Y 220.907,Z 408.056,A -85,B 0,C 180,E1 -23795.074,E2 -23795.074} C_VEL
LIN {X 0,Y 215.449,Z 477.189,A -85,B 0,C 180,E1 -23796.98,E2 -23796.98} C_VEL
LIN {X 0,Y 213.02,Z 492.886,A -85,B 0,C 180,E1 -23797.647,E2 -23797.647} C_VEL
LIN {X 0,Y 210.688,Z 503.913,A -85,B 0,C 180,E1 -23798.322,E2 -23798.322} C_VEL
LIN {X 0,Y 208.917,Z 509.51,A -85,B 0,C 180,E1 -23798.586,E2 -23798.586} C_VEL
LIN {X 0,Y 204.576,Z 518.373,A -85,B 0,C 180,E1 -23798.711,E2 -23798.711} C_VEL
LIN {X 0,Y 199.873,Z 527.096,A -85,B 0,C 180,E1 -23798.944,E2 -23798.944} C_VEL
LIN {X 0,Y 197.549,Z 532.254,A -85,B 0,C 180,E1 -23799.389,E2 -23799.389} C_VEL
LIN {X 0,Y 192.081,Z 545.775,A -85,B 0,C 180,E1 -23801.271,E2 -23801.271} C_VEL
LIN {X 0,Y 186.368,Z 557.998,A -85,B 0,C 180,E1 -23803.456,E2 -23803.456} C_VEL
LIN {X 0,Y 180.035,Z 569.835,A -85,B 0,C 180,E1 -23806.141,E2 -23806.141} C_VEL
LIN {X 0,Y 174.204,Z 579.803,A -85,B 0,C 180,E1 -23809.038,E2 -23809.038} C_VEL
LIN {X 0,Y 168.253,Z 589.237,A -85,B 0,C 180,E1 -23812.526,E2 -23812.526} C_VEL
LIN {X 0,Y 162.747,Z 597.718,A -85,B 0,C 180,E1 -23816.594,E2 -23816.594} C_VEL
LIN {X 0,Y 157.987,Z 604.461,A -85,B 0,C 180,E1 -23820.704,E2 -23820.704} C_VEL
LIN {X 0,Y 153.716,Z 610.698,A -85,B 0,C 180,E1 -23825.702,E2 -23825.702} C_VEL
LIN {X 0,Y 150.646,Z 615.531,A -85,B 0,C 180,E1 -23830.94,E2 -23830.94} C_VEL
LIN {X 0,Y 148.623,Z 619.079,A -85,B 0,C 180,E1 -23836.324,E2 -23836.324} C_VEL
LIN {X 0,Y 147.71,Z 621.422,A -85,B 0,C 180,E1 -23841.794,E2 -23841.794} C_VEL
LIN {X 0,Y 147.564,Z 622.605,A -85,B 0,C 180,E1 -23847.27,E2 -23847.27} C_VEL
LIN {X 0,Y 147.716,Z 622.765,A -85,B 0,C 180,E1 -23850,E2 -23850} C_VEL
LIN {X 0,Y 147.533,Z 622.139,A -85,B 0,C 180,E1 -23855.467,E2 -23855.467} C_VEL
LIN {X 0,Y 148.02,Z 620.357,A -85,B 0,C 180,E1 -23860.948,E2 -23860.948} C_VEL
LIN {X 0,Y 149.471,Z 617.401,A -85,B 0,C 180,E1 -23866.386,E2 -23866.386} C_VEL
LIN {X 0,Y 151.985,Z 613.205,A -85,B 0,C 180,E1 -23871.711,E2 -23871.711} C_VEL
LIN {X 0,Y 155.741,Z 607.664,A -85,B 0,C 180,E1 -23876.824,E2 -23876.824} C_VEL
LIN {X 0,Y 160.577,Z 600.626,A -85,B 0,C 180,E1 -23881.681,E2 -23881.681} C_VEL
LIN {X 0,Y 165.695,Z 593.108,A -85,B 0,C 180,E1 -23885.675,E2 -23885.675} C_VEL
LIN {X 0,Y 171.454,Z 584.047,A -85,B 0,C 180,E1 -23889.445,E2 -23889.445} C_VEL
LIN {X 0,Y 178.042,Z 573.167,A -85,B 0,C 180,E1 -23892.914,E2 -23892.914} C_VEL
LIN {X 0,Y 184.176,Z 561.97,A -85,B 0,C 180,E1 -23895.681,E2 -23895.681} C_VEL
LIN {X 0,Y 190.595,Z 548.937,A -85,B 0,C 180,E1 -23898.159,E2 -23898.159} C_VEL
LIN {X 0,Y 195.882,Z 536.211,A -85,B 0,C 180,E1 -23900.075,E2 -23900.075} C_VEL
LIN {X 0,Y 200.627,Z 522.954,A -85,B 0,C 180,E1 -23901.608,E2 -23901.608} C_VEL
LIN {X 0,Y 205.005,Z 508.451,A -85,B 0,C 180,E1 -23902.848,E2 -23902.848} C_VEL
LIN {X 0,Y 208.443,Z 493.406,A -85,B 0,C 180,E1 -23903.81,E2 -23903.81} C_VEL
LIN {X 0,Y 210.851,Z 478.307,A -85,B 0,C 180,E1 -23904.483,E2 -23904.483} C_VEL
LIN {X 0,Y 213.33,Z 450.556,A -85,B 0,C 180,E1 -23905.266,E2 -23905.266} C_VEL
LIN {X 0,Y 216.474,Z 410.504,A -85,B 0,C 180,E1 -23906.362,E2 -23906.362} C_VEL
LIN {X 0,Y 212.061,Z 399.307,A -85,B 0,C 180,E1 -23908.89,E2 -23908.89} C_VEL
LIN {X 0,Y 207.055,Z 388.254,A -85,B 0,C 180,E1 -23912.031,E2 -23912.031} C_VEL
LIN {X 0,Y 203.146,Z 380.603,A -85,B 0,C 180,E1 -23914.772,E2 -23914.772} C_VEL
LIN {X 0,Y 199.064,Z 374.276,A -85,B 0,C 180,E1 -23917.947,E2 -23917.947} C_VEL
LIN {X 0,Y 196.172,Z 370.135,A -85,B 0,C 180,E1 -23920.545,E2 -23920.545} C_VEL
LIN {X 0,Y 193.287,Z 365.946,A -85,B 0,C 180,E1 -23923.621,E2 -23923.621} C_VEL
LIN {X 0,Y 190.669,Z 362.273,A -85,B 0,C 180,E1 -23927.088,E2 -23927.088} C_VEL
LIN {X 0,Y 190.114,Z 361.278,A -85,B 0,C 180,E1 -23927.998,E2 -23927.998} C_VEL
LIN {X 0,Y 187.922,Z 358.768,A -85,B 0,C 180,E1 -23932.262,E2 -23932.262} C_VEL
LIN {X 0,Y 187.013,Z 356.189,A -85,B 0,C 180,E1 -23935.69,E2 -23935.69} C_VEL
LIN {X 0,Y 186.478,Z 355.786,A -85,B 0,C 180,E1 -23940,E2 -23940} C_VEL
LIN {X 0,Y 187.118,Z 356.434,A -85,B 0,C 180,E1 -23945.253,E2 -23945.253} C_VEL
LIN {X 0,Y 188.653,Z 360.017,A -85,B 0,C 180,E1 -23949.922,E2 -23949.922} C_VEL
LIN {X 0,Y 190.416,Z 361.685,A -85,B 0,C 180,E1 -23952.93,E2 -23952.93} C_VEL
LIN {X 0,Y 192.587,Z 365.255,A -85,B 0,C 180,E1 -23956.02,E2 -23956.02} C_VEL
LIN {X 0,Y 193.907,Z 366.802,A -85,B 0,C 180,E1 -23957.535,E2 -23957.535} C_VEL
LIN {X 0,Y 197.412,Z 371.877,A -85,B 0,C 180,E1 -23961.06,E2 -23961.06} C_VEL
LIN {X 0,Y 200.376,Z 376.333,A -85,B 0,C 180,E1 -23963.582,E2 -23963.582} C_VEL
LIN {X 0,Y 204.562,Z 382.765,A -85,B 0,C 180,E1 -23966.664,E2 -23966.664} C_VEL
LIN {X 0,Y 208.833,Z 390.047,A -85,B 0,C 180,E1 -23969.438,E2 -23969.438} C_VEL
LIN {X 0,Y 213.602,Z 398.776,A -85,B 0,C 180,E1 -23972.197,E2 -23972.197} C_VEL
LIN {X 0,Y 216.829,Z 405.155,A -85,B 0,C 180,E1 -23973.913,E2 -23973.913} C_VEL
LIN {X 0,Y 211.608,Z 469.685,A -85,B 0,C 180,E1 -23975.708,E2 -23975.708} C_VEL
LIN {X 0,Y 209.188,Z 485.234,A -85,B 0,C 180,E1 -23976.366,E2 -23976.366} C_VEL
LIN {X 0,Y 206.07,Z 499.932,A -85,B 0,C 180,E1 -23977.34,E2 -23977.34} C_VEL
LIN {X 0,Y 202.015,Z 514.507,A -85,B 0,C 180,E1 -23978.647,E2 -23978.647} C_VEL
LIN {X 0,Y 197.689,Z 527.378,A -85,B 0,C 180,E1 -23980.184,E2 -23980.184} C_VEL
LIN {X 0,Y 192.099,Z 541.001,A -85,B 0,C 180,E1 -23982.198,E2 -23982.198} C_VEL
LIN {X 0,Y 186.223,Z 553.401,A -85,B 0,C 180,E1 -23984.576,E2 -23984.576} C_VEL
LIN {X 0,Y 180.589,Z 563.785,A -85,B 0,C 180,E1 -23987.076,E2 -23987.076} C_VEL
LIN {X 0,Y 174.973,Z 573.411,A -85,B 0,C 180,E1 -23990.011,E2 -23990.011} C_VEL
LIN {X 0,Y 170.706,Z 580.361,A -85,B 0,C 180,E1 -23992.61,E2 -23992.61} C_VEL
LIN {X 0,Y 165.129,Z 588.61,A -85,B 0,C 180,E1 -23996.408,E2 -23996.408} C_VEL
LIN {X 0,Y 159.619,Z 596.354,A -85,B 0,C 180,E1 -24001.032,E2 -24001.032} C_VEL
LIN {X 0,Y 155.238,Z 602.507,A -85,B 0,C 180,E1 -24005.956,E2 -24005.956} C_VEL
LIN {X 0,Y 151.84,Z 607.253,A -85,B 0,C 180,E1 -24011.096,E2 -24011.096} C_VEL
LIN {X 0,Y 149.634,Z 610.718,A -85,B 0,C 180,E1 -24016.418,E2 -24016.418} C_VEL
LIN {X 0,Y 148.278,Z 613.004,A -85,B 0,C 180,E1 -24021.826,E2 -24021.826} C_VEL
LIN {X 0,Y 147.756,Z 614.163,A -85,B 0,C 180,E1 -24027.274,E2 -24027.274} C_VEL
LIN {X 0,Y 147.766,Z 614.316,A -85,B 0,C 180,E1 -24030,E2 -24030} C_VEL
LIN {X 0,Y 147.937,Z 613.755,A -85,B 0,C 180,E1 -24035.452,E2 -24035.452} C_VEL
LIN {X 0,Y 148.83,Z 612.081,A -85,B 0,C 180,E1 -24040.888,E2 -24040.888} C_VEL
LIN {X 0,Y 150.567,Z 609.255,A -85,B 0,C 180,E1 -24046.263,E2 -24046.263} C_VEL
LIN {X 0,Y 153.431,Z 605.2,A -85,B 0,C 180,E1 -24051.496,E2 -24051.496} C_VEL
LIN {X 0,Y 157.613,Z 599.352,A -85,B 0,C 180,E1 -24056.899,E2 -24056.899} C_VEL
LIN {X 0,Y 162.197,Z 592.956,A -85,B 0,C 180,E1 -24061.329,E2 -24061.329} C_VEL
LIN {X 0,Y 168.087,Z 584.383,A -85,B 0,C 180,E1 -24065.827,E2 -24065.827} C_VEL
LIN {X 0,Y 173.19,Z 576.669,A -85,B 0,C 180,E1 -24068.974,E2 -24068.974} C_VEL
LIN {X 0,Y 177.562,Z 569.312,A -85,B 0,C 180,E1 -24071.476,E2 -24071.476} C_VEL
LIN {X 0,Y 183.565,Z 558.806,A -85,B 0,C 180,E1 -24074.323,E2 -24074.323} C_VEL
LIN {X 0,Y 189.254,Z 547.492,A -85,B 0,C 180,E1 -24076.783,E2 -24076.783} C_VEL
LIN {X 0,Y 194.794,Z 535.189,A -85,B 0,C 180,E1 -24078.862,E2 -24078.862} C_VEL
LIN {X 0,Y 199.827,Z 521.734,A -85,B 0,C 180,E1 -24080.69,E2 -24080.69} C_VEL
LIN {X 0,Y 204.172,Z 507.878,A -85,B 0,C 180,E1 -24082.122,E2 -24082.122} C_VEL
LIN {X 0,Y 207.757,Z 493.432,A -85,B 0,C 180,E1 -24083.252,E2 -24083.252} C_VEL
LIN {X 0,Y 210.695,Z 477.572,A -85,B 0,C 180,E1 -24084.127,E2 -24084.127} C_VEL
LIN {X 0,Y 212.505,Z 462.248,A -85,B 0,C 180,E1 -24084.663,E2 -24084.663} C_VEL
LIN {X 0,Y 217.037,Z 405.339,A -85,B 0,C 180,E1 -24086.2,E2 -24086.2} C_VEL
LIN {X 0,Y 211.35,Z 394.284,A -85,B 0,C 180,E1 -24089.311,E2 -24089.311} C_VEL
LIN {X 0,Y 206.011,Z 385.008,A -85,B 0,C 180,E1 -24092.619,E2 -24092.619} C_VEL
LIN {X 0,Y 201.418,Z 377.758,A -85,B 0,C 180,E1 -24095.898,E2 -24095.898} C_VEL
LIN {X 0,Y 198.754,Z 373.803,A -85,B 0,C 180,E1 -24098.068,E2 -24098.068} C_VEL
LIN {X 0,Y 196.367,Z 370.285,A -85,B 0,C 180,E1 -24100.259,E2 -24100.259} C_VEL
LIN {X 0,Y 193.463,Z 366.078,A -85,B 0,C 180,E1 -24103.376,E2 -24103.376} C_VEL
LIN {X 0,Y 191.119,Z 362.959,A -85,B 0,C 180,E1 -24106.442,E2 -24106.442} C_VEL
LIN {X 0,Y 190.422,Z 361.466,A -85,B 0,C 180,E1 -24107.612,E2 -24107.612} C_VEL
LIN {X 0,Y 188.228,Z 359.196,A -85,B 0,C 180,E1 -24111.816,E2 -24111.816} C_VEL
LIN {X 0,Y 187.234,Z 356.309,A -85,B 0,C 180,E1 -24115.694,E2 -24115.694} C_VEL
LIN {X 0,Y 186.792,Z 355.956,A -85,B 0,C 180,E1 -24120,E2 -24120} C_VEL
LIN {X 0,Y 187.235,Z 356.464,A -85,B 0,C 180,E1 -24124.036,E2 -24124.036} C_VEL
LIN {X 0,Y 189.102,Z 360.416,A -85,B 0,C 180,E1 -24129.795,E2 -24129.795} C_VEL
LIN {X 0,Y 190.538,Z 361.782,A -85,B 0,C 180,E1 -24132.245,E2 -24132.245} C_VEL
LIN {X 0,Y 192.982,Z 365.625,A -85,B 0,C 180,E1 -24135.715,E2 -24135.715} C_VEL
LIN {X 0,Y 194.077,Z 366.975,A -85,B 0,C 180,E1 -24136.98,E2 -24136.98} C_VEL
LIN {X 0,Y 197.355,Z 371.665,A -85,B 0,C 180,E1 -24140.316,E2 -24140.316} C_VEL
LIN {X 0,Y 200.201,Z 375.91,A -85,B 0,C 180,E1 -24142.78,E2 -24142.78} C_VEL
LIN {X 0,Y 203.731,Z 381.37,A -85,B 0,C 180,E1 -24145.46,E2 -24145.46} C_VEL
LIN {X 0,Y 208.034,Z 390.131,A -85,B 0,C 180,E1 -24148.453,E2 -24148.453} C_VEL
LIN {X 0,Y 212.459,Z 400.064,A -85,B 0,C 180,E1 -24151.205,E2 -24151.205} C_VEL
LIN {X 0,Y 216.568,Z 410.366,A -85,B 0,C 180,E1 -24153.552,E2 -24153.552} C_VEL
LIN {X 0,Y 216.574,Z 412.389,A -85,B 0,C 180,E1 -24153.672,E2 -24153.672} C_VEL
LIN {X 0,Y 211.263,Z 476.995,A -85,B 0,C 180,E1 -24155.444,E2 -24155.444} C_VEL
LIN {X 0,Y 208.757,Z 492.692,A -85,B 0,C 180,E1 -24156.103,E2 -24156.103} C_VEL
LIN {X 0,Y 205.295,Z 507.922,A -85,B 0,C 180,E1 -24157.056,E2 -24157.056} C_VEL
LIN {X 0,Y 201.277,Z 521.649,A -85,B 0,C 180,E1 -24158.223,E2 -24158.223} C_VEL
LIN {X 0,Y 197.549,Z 532.254,A -85,B 0,C 180,E1 -24159.389,E2 -24159.389} C_VEL
LIN {X 0,Y 195.144,Z 537.41,A -85,B 0,C 180,E1 -24159.896,E2 -24159.896} C_VEL
LIN {X 0,Y 189.857,Z 545.547,A -85,B 0,C 180,E1 -24160.456,E2 -24160.456} C_VEL
LIN {X 0,Y 184.265,Z 553.44,A -85,B 0,C 180,E1 -24161.147,E2 -24161.147} C_VEL
LIN {X 0,Y 181.415,Z 558.043,A -85,B 0,C 180,E1 -24161.874,E2 -24161.874} C_VEL
LIN {X 0,Y 174.95,Z 569.634,A -85,B 0,C 180,E1 -24164.518,E2 -24164.518} C_VEL
LIN {X 0,Y 168.86,Z 579.601,A -85,B 0,C 180,E1 -24167.444,E2 -24167.444} C_VEL
LIN {X 0,Y 163.181,Z 588.222,A -85,B 0,C 180,E1 -24170.634,E2 -24170.634} C_VEL
LIN {X 0,Y 157.583,Z 596.434,A -85,B 0,C 180,E1 -24174.566,E2 -24174.566} C_VEL
LIN {X 0,Y 151.776,Z 604.258,A -85,B 0,C 180,E1 -24179.38,E2 -24179.38} C_VEL
LIN {X 0,Y 147.219,Z 610.494,A -85,B 0,C 180,E1 -24184.556,E2 -24184.556} C_VEL
LIN {X 0,Y 143.877,Z 615.327,A -85,B 0,C 180,E1 -24190.006,E2 -24190.006} C_VEL
LIN {X 0,Y 141.667,Z 618.875,A -85,B 0,C 180,E1 -24195.638,E2 -24195.638} C_VEL
LIN {X 0,Y 140.65,Z 621.218,A -85,B 0,C 180,E1 -24201.379,E2 -24201.379} C_VEL
LIN {X 0,Y 140.481,Z 622.403,A -85,B 0,C 180,E1 -24207.132,E2 -24207.132} C_VEL
LIN {X 0,Y 140.568,Z 622.528,A -85,B 0,C 180,E1 -24210.644,E2 -24210.644} C_VEL
LIN {X 0,Y 140.441,Z 621.935,A -85,B 0,C 180,E1 -24215.744,E2 -24215.744} C_VEL
LIN {X 0,Y 141.018,Z 620.152,A -85,B 0,C 180,E1 -24221.499,E2 -24221.499} C_VEL
LIN {X 0,Y 142.624,Z 617.195,A -85,B 0,C 180,E1 -24227.197,E2 -24227.197} C_VEL
LIN {X 0,Y 145.31,Z 612.997,A -85,B 0,C 180,E1 -24232.763,E2 -24232.763} C_VEL
LIN {X 0,Y 149.368,Z 607.457,A -85,B 0,C 180,E1 -24238.067,E2 -24238.067} C_VEL
LIN {X 0,Y 154.529,Z 600.419,A -85,B 0,C 180,E1 -24243.076,E2 -24243.076} C_VEL
LIN {X 0,Y 159.925,Z 592.901,A -85,B 0,C 180,E1 -24247.174,E2 -24247.174} C_VEL
LIN {X 0,Y 165.982,Z 583.84,A -85,B 0,C 180,E1 -24251.017,E2 -24251.017} C_VEL
LIN {X 0,Y 172.883,Z 572.96,A -85,B 0,C 180,E1 -24254.525,E2 -24254.525} C_VEL
LIN {X 0,Y 179.275,Z 561.763,A -85,B 0,C 180,E1 -24257.309,E2 -24257.309} C_VEL
LIN {X 0,Y 185.722,Z 549.125,A -85,B 0,C 180,E1 -24259.732,E2 -24259.732} C_VEL
LIN {X 0,Y 191.382,Z 536.002,A -85,B 0,C 180,E1 -24261.713,E2 -24261.713} C_VEL
LIN {X 0,Y 196.291,Z 522.746,A -85,B 0,C 180,E1 -24263.234,E2 -24263.234} C_VEL
LIN {X 0,Y 200.783,Z 508.24,A -85,B 0,C 180,E1 -24264.468,E2 -24264.468} C_VEL
LIN {X 0,Y 204.322,Z 493.193,A -85,B 0,C 180,E1 -24265.421,E2 -24265.421} C_VEL
LIN {X 0,Y 206.798,Z 478.135,A -85,B 0,C 180,E1 -24266.084,E2 -24266.084} C_VEL
LIN {X 0,Y 209.352,Z 450.582,A -85,B 0,C 180,E1 -24266.854,E2 -24266.854} C_VEL
LIN {X 0,Y 212.37,Z 413.147,A -85,B 0,C 180,E1 -24267.886,E2 -24267.886} C_VEL
LIN {X 0,Y 208,Z 401.993,A -85,B 0,C 180,E1 -24270.595,E2 -24270.595} C_VEL
LIN {X 0,Y 203.75,Z 392.398,A -85,B 0,C 180,E1 -24273.497,E2 -24273.497} C_VEL
LIN {X 0,Y 200.653,Z 386.143,A -85,B 0,C 180,E1 -24275.836,E2 -24275.836} C_VEL
LIN {X 0,Y 196.882,Z 380.245,A -85,B 0,C 180,E1 -24278.956,E2 -24278.956} C_VEL
LIN {X 0,Y 194.568,Z 376.736,A -85,B 0,C 180,E1 -24281.166,E2 -24281.166} C_VEL
LIN {X 0,Y 191.775,Z 372.551,A -85,B 0,C 180,E1 -24284.302,E2 -24284.302} C_VEL
LIN {X 0,Y 189.303,Z 368.815,A -85,B 0,C 180,E1 -24287.81,E2 -24287.81} C_VEL
LIN {X 0,Y 188.923,Z 368.145,A -85,B 0,C 180,E1 -24288.466,E2 -24288.466} C_VEL
LIN {X 0,Y 186.851,Z 365.582,A -85,B 0,C 180,E1 -24292.775,E2 -24292.775} C_VEL
LIN {X 0,Y 186.144,Z 363.287,A -85,B 0,C 180,E1 -24295.67,E2 -24295.67} C_VEL
LIN {X 0,Y 185.613,Z 362.835,A -85,B 0,C 180,E1 -24300,E2 -24300} C_VEL
LIN {X 0,Y 186.176,Z 363.516,A -85,B 0,C 180,E1 -24305.008,E2 -24305.008} C_VEL
LIN {X 0,Y 187.661,Z 367.011,A -85,B 0,C 180,E1 -24309.702,E2 -24309.702} C_VEL
LIN {X 0,Y 189.194,Z 368.558,A -85,B 0,C 180,E1 -24312.442,E2 -24312.442} C_VEL
LIN {X 0,Y 191.412,Z 372.196,A -85,B 0,C 180,E1 -24315.711,E2 -24315.711} C_VEL
LIN {X 0,Y 192.475,Z 373.531,A -85,B 0,C 180,E1 -24316.985,E2 -24316.985} C_VEL
LIN {X 0,Y 195.734,Z 378.44,A -85,B 0,C 180,E1 -24320.424,E2 -24320.424} C_VEL
LIN {X 0,Y 198.779,Z 383.194,A -85,B 0,C 180,E1 -24323.124,E2 -24323.124} C_VEL
LIN {X 0,Y 202.737,Z 389.609,A -85,B 0,C 180,E1 -24326.156,E2 -24326.156} C_VEL
LIN {X 0,Y 207.48,Z 398.01,A -85,B 0,C 180,E1 -24329.323,E2 -24329.323} C_VEL
LIN {X 0,Y 212.672,Z 408.27,A -85,B 0,C 180,E1 -24332.388,E2 -24332.388} C_VEL
LIN {X 0,Y 207.524,Z 470.149,A -85,B 0,C 180,E1 -24334.13,E2 -24334.13} C_VEL
LIN {X 0,Y 205.072,Z 485.447,A -85,B 0,C 180,E1 -24334.774,E2 -24334.774} C_VEL
LIN {X 0,Y 201.844,Z 500.143,A -85,B 0,C 180,E1 -24335.738,E2 -24335.738} C_VEL
LIN {X 0,Y 197.667,Z 514.716,A -85,B 0,C 180,E1 -24337.043,E2 -24337.043} C_VEL
LIN {X 0,Y 193.08,Z 527.881,A -85,B 0,C 180,E1 -24338.615,E2 -24338.615} C_VEL
LIN {X 0,Y 187.412,Z 541.208,A -85,B 0,C 180,E1 -24340.592,E2 -24340.592} C_VEL
LIN {X 0,Y 181.295,Z 553.608,A -85,B 0,C 180,E1 -24342.973,E2 -24342.973} C_VEL
LIN {X 0,Y 175.456,Z 563.991,A -85,B 0,C 180,E1 -24345.497,E2 -24345.497} C_VEL
LIN {X 0,Y 169.554,Z 573.618,A -85,B 0,C 180,E1 -24348.457,E2 -24348.457} C_VEL
LIN {X 0,Y 165.114,Z 580.566,A -85,B 0,C 180,E1 -24351.111,E2 -24351.111} C_VEL
LIN {X 0,Y 159.232,Z 588.816,A -85,B 0,C 180,E1 -24354.987,E2 -24354.987} C_VEL
LIN {X 0,Y 153.433,Z 596.559,A -85,B 0,C 180,E1 -24359.746,E2 -24359.746} C_VEL
LIN {X 0,Y 148.739,Z 602.713,A -85,B 0,C 180,E1 -24364.834,E2 -24364.834} C_VEL
LIN {X 0,Y 145.108,Z 607.458,A -85,B 0,C 180,E1 -24370.183,E2 -24370.183} C_VEL
LIN {X 0,Y 142.704,Z 610.923,A -85,B 0,C 180,E1 -24375.745,E2 -24375.745} C_VEL
LIN {X 0,Y 141.254,Z 613.207,A -85,B 0,C 180,E1 -24381.416,E2 -24381.416} C_VEL
LIN {X 0,Y 140.677,Z 614.366,A -85,B 0,C 180,E1 -24387.137,E2 -24387.137} C_VEL
LIN {X 0,Y 140.653,Z 614.419,A -85,B 0,C 180,E1 -24392.077,E2 -24392.077} C_VEL
LIN {X 0,Y 140.865,Z 613.958,A -85,B 0,C 180,E1 -24395.727,E2 -24395.727} C_VEL
LIN {X 0,Y 141.838,Z 612.285,A -85,B 0,C 180,E1 -24401.431,E2 -24401.431} C_VEL
LIN {X 0,Y 143.732,Z 609.459,A -85,B 0,C 180,E1 -24407.06,E2 -24407.06} C_VEL
LIN {X 0,Y 146.815,Z 605.403,A -85,B 0,C 180,E1 -24412.516,E2 -24412.516} C_VEL
LIN {X 0,Y 151.063,Z 599.861,A -85,B 0,C 180,E1 -24417.877,E2 -24417.877} C_VEL
LIN {X 0,Y 156.135,Z 593.159,A -85,B 0,C 180,E1 -24422.693,E2 -24422.693} C_VEL
LIN {X 0,Y 162.361,Z 584.584,A -85,B 0,C 180,E1 -24427.3,E2 -24427.3} C_VEL
LIN {X 0,Y 167.689,Z 576.871,A -85,B 0,C 180,E1 -24430.511,E2 -24430.511} C_VEL
LIN {X 0,Y 172.362,Z 569.409,A -85,B 0,C 180,E1 -24433.074,E2 -24433.074} C_VEL
LIN {X 0,Y 178.545,Z 559.007,A -85,B 0,C 180,E1 -24435.918,E2 -24435.918} C_VEL
LIN {X 0,Y 184.467,Z 547.692,A -85,B 0,C 180,E1 -24438.389,E2 -24438.389} C_VEL
LIN {X 0,Y 190.208,Z 535.387,A -85,B 0,C 180,E1 -24440.47,E2 -24440.47} C_VEL
LIN {X 0,Y 195.536,Z 521.591,A -85,B 0,C 180,E1 -24442.337,E2 -24442.337} C_VEL
LIN {X 0,Y 200.229,Z 506.898,A -85,B 0,C 180,E1 -24443.83,E2 -24443.83} C_VEL
LIN {X 0,Y 203.896,Z 492.248,A -85,B 0,C 180,E1 -24444.945,E2 -24444.945} C_VEL
LIN {X 0,Y 206.787,Z 476.67,A -85,B 0,C 180,E1 -24445.762,E2 -24445.762} C_VEL
LIN {X 0,Y 208.627,Z 460.551,A -85,B 0,C 180,E1 -24446.311,E2 -24446.311} C_VEL
LIN {X 0,Y 212.903,Z 408.443,A -85,B 0,C 180,E1 -24447.718,E2 -24447.718} C_VEL
LIN {X 0,Y 207.482,Z 397.759,A -85,B 0,C 180,E1 -24450.931,E2 -24450.931} C_VEL
LIN {X 0,Y 202.713,Z 389.393,A -85,B 0,C 180,E1 -24454.138,E2 -24454.138} C_VEL
LIN {X 0,Y 198.854,Z 383.165,A -85,B 0,C 180,E1 -24457.122,E2 -24457.122} C_VEL
LIN {X 0,Y 196.506,Z 379.567,A -85,B 0,C 180,E1 -24459.181,E2 -24459.181} C_VEL
LIN {X 0,Y 194.74,Z 376.841,A -85,B 0,C 180,E1 -24460.909,E2 -24460.909} C_VEL
LIN {X 0,Y 192.061,Z 372.784,A -85,B 0,C 180,E1 -24463.935,E2 -24463.935} C_VEL
LIN {X 0,Y 189.745,Z 369.487,A -85,B 0,C 180,E1 -24467.159,E2 -24467.159} C_VEL
LIN {X 0,Y 189.148,Z 368.299,A -85,B 0,C 180,E1 -24468.208,E2 -24468.208} C_VEL
LIN {X 0,Y 187.115,Z 365.931,A -85,B 0,C 180,E1 -24472.446,E2 -24472.446} C_VEL
LIN {X 0,Y 186.26,Z 363.29,A -85,B 0,C 180,E1 -24476.214,E2 -24476.214} C_VEL
LIN {X 0,Y 186.066,Z 363.136,A -85,B 0,C 180,E1 -24482.164,E2 -24482.164} C_VEL
LIN {X 0,Y 186.333,Z 363.574,A -85,B 0,C 180,E1 -24483.92,E2 -24483.92} C_VEL
LIN {X 0,Y 188.154,Z 367.467,A -85,B 0,C 180,E1 -24489.676,E2 -24489.676} C_VEL
LIN {X 0,Y 189.412,Z 368.828,A -85,B 0,C 180,E1 -24491.911,E2 -24491.911} C_VEL
LIN {X 0,Y 191.962,Z 372.727,A -85,B 0,C 180,E1 -24495.596,E2 -24495.596} C_VEL
LIN {X 0,Y 195.624,Z 378.14,A -85,B 0,C 180,E1 -24499.614,E2 -24499.614} C_VEL
LIN {X 0,Y 198.368,Z 382.413,A -85,B 0,C 180,E1 -24502.113,E2 -24502.113} C_VEL
LIN {X 0,Y 201.365,Z 387.163,A -85,B 0,C 180,E1 -24504.509,E2 -24504.509} C_VEL
LIN {X 0,Y 205.338,Z 395.61,A -85,B 0,C 180,E1 -24507.451,E2 -24507.451} C_VEL
LIN {X 0,Y 209.328,Z 404.986,A -85,B 0,C 180,E1 -24510.1,E2 -24510.1} C_VEL
LIN {X 0,Y 212.555,Z 413.323,A -85,B 0,C 180,E1 -24512.079,E2 -24512.079} C_VEL
LIN {X 0,Y 207.211,Z 476.923,A -85,B 0,C 180,E1 -24513.849,E2 -24513.849} C_VEL
LIN {X 0,Y 204.659,Z 492.499,A -85,B 0,C 180,E1 -24514.499,E2 -24514.499} C_VEL
LIN {X 0,Y 201.102,Z 507.726,A -85,B 0,C 180,E1 -24515.443,E2 -24515.443} C_VEL
LIN {X 0,Y 196.946,Z 521.451,A -85,B 0,C 180,E1 -24516.593,E2 -24516.593} C_VEL
LIN {X 0,Y 192.002,Z 534.901,A -85,B 0,C 180,E1 -24518.098,E2 -24518.098} C_VEL
LIN {X 0,Y 186.681,Z 547.36,A -85,B 0,C 180,E1 -24519.927,E2 -24519.927} C_VEL
LIN {X 0,Y 181.415,Z 558.043,A -85,B 0,C 180,E1 -24521.874,E2 -24521.874} C_VEL
LIN {X 0,Y 178.482,Z 562.589,A -85,B 0,C 180,E1 -24522.661,E2 -24522.661} C_VEL
LIN {X 0,Y 172.353,Z 569.68,A -85,B 0,C 180,E1 -24523.703,E2 -24523.703} C_VEL
LIN {X 0,Y 166.109,Z 576.434,A -85,B 0,C 180,E1 -24524.948,E2 -24524.948} C_VEL
LIN {X 0,Y 163.051,Z 580.305,A -85,B 0,C 180,E1 -24526.063,E2 -24526.063} C_VEL
LIN {X 0,Y 156.264,Z 589.992,A -85,B 0,C 180,E1 -24529.869,E2 -24529.869} C_VEL
LIN {X 0,Y 150.188,Z 598.327,A -85,B 0,C 180,E1 -24534.203,E2 -24534.203} C_VEL
LIN {X 0,Y 144.31,Z 605.73,A -85,B 0,C 180,E1 -24539.247,E2 -24539.247} C_VEL
LIN {X 0,Y 139.39,Z 612.044,A -85,B 0,C 180,E1 -24545.168,E2 -24545.168} C_VEL
LIN {X 0,Y 137.158,Z 615.122,A -85,B 0,C 180,E1 -24548.981,E2 -24548.981} C_VEL
LIN {X 0,Y 134.736,Z 618.67,A -85,B 0,C 180,E1 -24554.882,E2 -24554.882} C_VEL
LIN {X 0,Y 133.589,Z 621.014,A -85,B 0,C 180,E1 -24560.919,E2 -24560.919} C_VEL
LIN {X 0,Y 133.389,Z 622.2,A -85,B 0,C 180,E1 -24566.98,E2 -24566.98} C_VEL
LIN {X 0,Y 133.531,Z 622.359,A -85,B 0,C 180,E1 -24570,E2 -24570} C_VEL
LIN {X 0,Y 133.374,Z 621.732,A -85,B 0,C 180,E1 -24576.049,E2 -24576.049} C_VEL
LIN {X 0,Y 134.003,Z 619.947,A -85,B 0,C 180,E1 -24582.109,E2 -24582.109} C_VEL
LIN {X 0,Y 135.782,Z 616.99,A -85,B 0,C 180,E1 -24588.092,E2 -24588.092} C_VEL
LIN {X 0,Y 138.695,Z 612.79,A -85,B 0,C 180,E1 -24593.914,E2 -24593.914} C_VEL
LIN {X 0,Y 143.06,Z 607.25,A -85,B 0,C 180,E1 -24599.423,E2 -24599.423} C_VEL
LIN {X 0,Y 148.59,Z 600.213,A -85,B 0,C 180,E1 -24604.58,E2 -24604.58} C_VEL
LIN {X 0,Y 154.279,Z 592.694,A -85,B 0,C 180,E1 -24608.781,E2 -24608.781} C_VEL
LIN {X 0,Y 160.646,Z 583.633,A -85,B 0,C 180,E1 -24612.694,E2 -24612.694} C_VEL
LIN {X 0,Y 167.874,Z 572.753,A -85,B 0,C 180,E1 -24616.232,E2 -24616.232} C_VEL
LIN {X 0,Y 174.517,Z 561.556,A -85,B 0,C 180,E1 -24619.031,E2 -24619.031} C_VEL
LIN {X 0,Y 180.978,Z 549.342,A -85,B 0,C 180,E1 -24621.378,E2 -24621.378} C_VEL
LIN {X 0,Y 186.423,Z 537.225,A -85,B 0,C 180,E1 -24623.234,E2 -24623.234} C_VEL
LIN {X 0,Y 191.482,Z 524.306,A -85,B 0,C 180,E1 -24624.748,E2 -24624.748} C_VEL
LIN {X 0,Y 196.077,Z 510.289,A -85,B 0,C 180,E1 -24625.98,E2 -24625.98} C_VEL
LIN {X 0,Y 199.892,Z 495.271,A -85,B 0,C 180,E1 -24626.961,E2 -24626.961} C_VEL
LIN {X 0,Y 202.664,Z 479.811,A -85,B 0,C 180,E1 -24627.67,E2 -24627.67} C_VEL
LIN {X 0,Y 204.798,Z 459.174,A -85,B 0,C 180,E1 -24628.278,E2 -24628.278} C_VEL
LIN {X 0,Y 208.442,Z 416.081,A -85,B 0,C 180,E1 -24629.44,E2 -24629.44} C_VEL
LIN {X 0,Y 204.958,Z 406.837,A -85,B 0,C 180,E1 -24631.775,E2 -24631.775} C_VEL
LIN {X 0,Y 201.274,Z 398.105,A -85,B 0,C 180,E1 -24634.47,E2 -24634.47} C_VEL
LIN {X 0,Y 198.315,Z 391.916,A -85,B 0,C 180,E1 -24636.85,E2 -24636.85} C_VEL
LIN {X 0,Y 195.062,Z 386.609,A -85,B 0,C 180,E1 -24639.709,E2 -24639.709} C_VEL
LIN {X 0,Y 192.927,Z 383.206,A -85,B 0,C 180,E1 -24641.867,E2 -24641.867} C_VEL
LIN {X 0,Y 190.376,Z 379.266,A -85,B 0,C 180,E1 -24644.884,E2 -24644.884} C_VEL
LIN {X 0,Y 187.824,Z 375.08,A -85,B 0,C 180,E1 -24648.808,E2 -24648.808} C_VEL
LIN {X 0,Y 185.819,Z 372.464,A -85,B 0,C 180,E1 -24653.212,E2 -24653.212} C_VEL
LIN {X 0,Y 185.157,Z 370.271,A -85,B 0,C 180,E1 -24656.192,E2 -24656.192} C_VEL
LIN {X 0,Y 184.747,Z 369.884,A -85,B 0,C 180,E1 -24660,E2 -24660} C_VEL
LIN {X 0,Y 185.218,Z 370.485,A -85,B 0,C 180,E1 -24664.625,E2 -24664.625} C_VEL
LIN {X 0,Y 186.669,Z 374.025,A -85,B 0,C 180,E1 -24669.481,E2 -24669.481} C_VEL
LIN {X 0,Y 188.062,Z 375.549,A -85,B 0,C 180,E1 -24672.079,E2 -24672.079} C_VEL
LIN {X 0,Y 190.243,Z 379.137,A -85,B 0,C 180,E1 -24675.398,E2 -24675.398} C_VEL
LIN {X 0,Y 191.26,Z 380.667,A -85,B 0,C 180,E1 -24676.683,E2 -24676.683} C_VEL
LIN {X 0,Y 193.848,Z 384.618,A -85,B 0,C 180,E1 -24679.539,E2 -24679.539} C_VEL
LIN {X 0,Y 196.639,Z 389.18,A -85,B 0,C 180,E1 -24682.18,E2 -24682.18} C_VEL
LIN {X 0,Y 200.581,Z 395.786,A -85,B 0,C 180,E1 -24685.374,E2 -24685.374} C_VEL
LIN {X 0,Y 205.33,Z 404.596,A -85,B 0,C 180,E1 -24688.703,E2 -24688.703} C_VEL
LIN {X 0,Y 208.764,Z 411.664,A -85,B 0,C 180,E1 -24690.865,E2 -24690.865} C_VEL
LIN {X 0,Y 203.7,Z 469.906,A -85,B 0,C 180,E1 -24692.467,E2 -24692.467} C_VEL
LIN {X 0,Y 201.123,Z 485.659,A -85,B 0,C 180,E1 -24693.119,E2 -24693.119} C_VEL
LIN {X 0,Y 197.778,Z 500.354,A -85,B 0,C 180,E1 -24694.067,E2 -24694.067} C_VEL
LIN {X 0,Y 193.47,Z 514.925,A -85,B 0,C 180,E1 -24695.364,E2 -24695.364} C_VEL
LIN {X 0,Y 188.589,Z 528.448,A -85,B 0,C 180,E1 -24696.974,E2 -24696.974} C_VEL
LIN {X 0,Y 182.877,Z 541.414,A -85,B 0,C 180,E1 -24698.905,E2 -24698.905} C_VEL
LIN {X 0,Y 176.515,Z 553.815,A -85,B 0,C 180,E1 -24701.28,E2 -24701.28} C_VEL
LIN {X 0,Y 170.46,Z 564.197,A -85,B 0,C 180,E1 -24703.822,E2 -24703.822} C_VEL
LIN {X 0,Y 164.277,Z 573.825,A -85,B 0,C 180,E1 -24706.805,E2 -24706.805} C_VEL
LIN {X 0,Y 158.686,Z 582.033,A -85,B 0,C 180,E1 -24710.046,E2 -24710.046} C_VEL
LIN {X 0,Y 152.638,Z 590.105,A -85,B 0,C 180,E1 -24714.053,E2 -24714.053} C_VEL
LIN {X 0,Y 147.305,Z 596.764,A -85,B 0,C 180,E1 -24718.345,E2 -24718.345} C_VEL
LIN {X 0,Y 142.31,Z 602.918,A -85,B 0,C 180,E1 -24723.612,E2 -24723.612} C_VEL
LIN {X 0,Y 138.424,Z 607.663,A -85,B 0,C 180,E1 -24729.183,E2 -24729.183} C_VEL
LIN {X 0,Y 135.807,Z 611.127,A -85,B 0,C 180,E1 -24735.005,E2 -24735.005} C_VEL
LIN {X 0,Y 134.217,Z 613.411,A -85,B 0,C 180,E1 -24740.962,E2 -24740.962} C_VEL
LIN {X 0,Y 133.602,Z 614.568,A -85,B 0,C 180,E1 -24746.985,E2 -24746.985} C_VEL
LIN {X 0,Y 133.56,Z 614.673,A -85,B 0,C 180,E1 -24751.167,E2 -24751.167} C_VEL
LIN {X 0,Y 133.807,Z 614.16,A -85,B 0,C 180,E1 -24756.03,E2 -24756.03} C_VEL
LIN {X 0,Y 134.874,Z 612.488,A -85,B 0,C 180,E1 -24762.03,E2 -24762.03} C_VEL
LIN {X 0,Y 136.914,Z 609.662,A -85,B 0,C 180,E1 -24767.938,E2 -24767.938} C_VEL
LIN {X 0,Y 140.255,Z 605.606,A -85,B 0,C 180,E1 -24773.632,E2 -24773.632} C_VEL
LIN {X 0,Y 144.659,Z 600.225,A -85,B 0,C 180,E1 -24779.066,E2 -24779.066} C_VEL
LIN {X 0,Y 150.183,Z 593.361,A -85,B 0,C 180,E1 -24784.162,E2 -24784.162} C_VEL
LIN {X 0,Y 155.871,Z 585.98,A -85,B 0,C 180,E1 -24788.313,E2 -24788.313} C_VEL
LIN {X 0,Y 161.371,Z 578.489,A -85,B 0,C 180,E1 -24791.572,E2 -24791.572} C_VEL
LIN {X 0,Y 166.188,Z 571.226,A -85,B 0,C 180,E1 -24794.246,E2 -24794.246} C_VEL
LIN {X 0,Y 172.568,Z 561.084,A -85,B 0,C 180,E1 -24797.142,E2 -24797.142} C_VEL
LIN {X 0,Y 179.245,Z 549.008,A -85,B 0,C 180,E1 -24799.867,E2 -24799.867} C_VEL
LIN {X 0,Y 185.16,Z 536.888,A -85,B 0,C 180,E1 -24801.959,E2 -24801.959} C_VEL
LIN {X 0,Y 190.415,Z 524.026,A -85,B 0,C 180,E1 -24803.75,E2 -24803.75} C_VEL
LIN {X 0,Y 194.876,Z 511.146,A -85,B 0,C 180,E1 -24805.128,E2 -24805.128} C_VEL
LIN {X 0,Y 198.667,Z 497.714,A -85,B 0,C 180,E1 -24806.233,E2 -24806.233} C_VEL
LIN {X 0,Y 201.796,Z 483.136,A -85,B 0,C 180,E1 -24807.128,E2 -24807.128} C_VEL
LIN {X 0,Y 204.11,Z 467.79,A -85,B 0,C 180,E1 -24807.738,E2 -24807.738} C_VEL
LIN {X 0,Y 208.95,Z 411.809,A -85,B 0,C 180,E1 -24809.266,E2 -24809.266} C_VEL
LIN {X 0,Y 204.49,Z 402.785,A -85,B 0,C 180,E1 -24812.114,E2 -24812.114} C_VEL
LIN {X 0,Y 199.87,Z 394.304,A -85,B 0,C 180,E1 -24815.466,E2 -24815.466} C_VEL
LIN {X 0,Y 195.519,Z 387.09,A -85,B 0,C 180,E1 -24819.181,E2 -24819.181} C_VEL
LIN {X 0,Y 192.991,Z 383.185,A -85,B 0,C 180,E1 -24821.728,E2 -24821.728} C_VEL
LIN {X 0,Y 190.546,Z 379.361,A -85,B 0,C 180,E1 -24824.665,E2 -24824.665} C_VEL
LIN {X 0,Y 188.38,Z 376.002,A -85,B 0,C 180,E1 -24827.92,E2 -24827.92} C_VEL
LIN {X 0,Y 187.819,Z 375.072,A -85,B 0,C 180,E1 -24828.944,E2 -24828.944} C_VEL
LIN {X 0,Y 185.833,Z 372.264,A -85,B 0,C 180,E1 -24833.746,E2 -24833.746} C_VEL
LIN {X 0,Y 185.393,Z 370.368,A -85,B 0,C 180,E1 -24836.196,E2 -24836.196} C_VEL
LIN {X 0,Y 185.064,Z 370.036,A -85,B 0,C 180,E1 -24840,E2 -24840} C_VEL
LIN {X 0,Y 185.392,Z 370.521,A -85,B 0,C 180,E1 -24843.532,E2 -24843.532} C_VEL
LIN {X 0,Y 187.291,Z 374.605,A -85,B 0,C 180,E1 -24849.721,E2 -24849.721} C_VEL
LIN {X 0,Y 188.203,Z 375.648,A -85,B 0,C 180,E1 -24851.4,E2 -24851.4} C_VEL
LIN {X 0,Y 190.735,Z 379.606,A -85,B 0,C 180,E1 -24855.22,E2 -24855.22} C_VEL
LIN {X 0,Y 194.045,Z 384.814,A -85,B 0,C 180,E1 -24859.024,E2 -24859.024} C_VEL
LIN {X 0,Y 196.802,Z 389.282,A -85,B 0,C 180,E1 -24861.643,E2 -24861.643} C_VEL
LIN {X 0,Y 199.271,Z 393.447,A -85,B 0,C 180,E1 -24863.718,E2 -24863.718} C_VEL
LIN {X 0,Y 203.195,Z 402.217,A -85,B 0,C 180,E1 -24866.782,E2 -24866.782} C_VEL
LIN {X 0,Y 207.481,Z 413.02,A -85,B 0,C 180,E1 -24869.765,E2 -24869.765} C_VEL
LIN {X 0,Y 208.598,Z 416.07,A -85,B 0,C 180,E1 -24870.496,E2 -24870.496} C_VEL
LIN {X 0,Y 203.44,Z 476.103,A -85,B 0,C 180,E1 -24872.172,E2 -24872.172} C_VEL
LIN {X 0,Y 200.847,Z 491.7,A -85,B 0,C 180,E1 -24872.794,E2 -24872.794} C_VEL
LIN {X 0,Y 197.072,Z 507.53,A -85,B 0,C 180,E1 -24873.763,E2 -24873.763} C_VEL
LIN {X 0,Y 192.801,Z 521.254,A -85,B 0,C 180,E1 -24874.9,E2 -24874.9} C_VEL
LIN {X 0,Y 187.699,Z 534.702,A -85,B 0,C 180,E1 -24876.39,E2 -24876.39} C_VEL
LIN {X 0,Y 182.162,Z 547.159,A -85,B 0,C 180,E1 -24878.197,E2 -24878.197} C_VEL
LIN {X 0,Y 175.693,Z 559.742,A -85,B 0,C 180,E1 -24880.535,E2 -24880.535} C_VEL
LIN {X 0,Y 168.929,Z 571.222,A -85,B 0,C 180,E1 -24883.278,E2 -24883.278} C_VEL
LIN {X 0,Y 163.051,Z 580.305,A -85,B 0,C 180,E1 -24886.063,E2 -24886.063} C_VEL
LIN {X 0,Y 159.978,Z 584.086,A -85,B 0,C 180,E1 -24887.265,E2 -24887.265} C_VEL
LIN {X 0,Y 153.574,Z 589.905,A -85,B 0,C 180,E1 -24889.026,E2 -24889.026} C_VEL
LIN {X 0,Y 147.198,Z 595.313,A -85,B 0,C 180,E1 -24891.05,E2 -24891.05} C_VEL
LIN {X 0,Y 144.247,Z 598.334,A -85,B 0,C 180,E1 -24892.665,E2 -24892.665} C_VEL
LIN {X 0,Y 138.201,Z 605.526,A -85,B 0,C 180,E1 -24897.728,E2 -24897.728} C_VEL
LIN {X 0,Y 133.187,Z 611.537,A -85,B 0,C 180,E1 -24903.521,E2 -24903.521} C_VEL
LIN {X 0,Y 130.496,Z 614.918,A -85,B 0,C 180,E1 -24907.853,E2 -24907.853} C_VEL
LIN {X 0,Y 127.829,Z 618.466,A -85,B 0,C 180,E1 -24914.045,E2 -24914.045} C_VEL
LIN {X 0,Y 126.551,Z 620.811,A -85,B 0,C 180,E1 -24920.41,E2 -24920.41} C_VEL
LIN {X 0,Y 126.294,Z 621.996,A -85,B 0,C 180,E1 -24926.81,E2 -24926.81} C_VEL
LIN {X 0,Y 126.427,Z 622.156,A -85,B 0,C 180,E1 -24930,E2 -24930} C_VEL
LIN {X 0,Y 126.293,Z 621.99,A -85,B 0,C 180,E1 -24933.19,E2 -24933.19} C_VEL
LIN {X 0,Y 126.53,Z 620.779,A -85,B 0,C 180,E1 -24939.592,E2 -24939.592} C_VEL
LIN {X 0,Y 127.805,Z 618.411,A -85,B 0,C 180,E1 -24945.959,E2 -24945.959} C_VEL
LIN {X 0,Y 130.44,Z 614.846,A -85,B 0,C 180,E1 -24952.157,E2 -24952.157} C_VEL
LIN {X 0,Y 134.394,Z 609.992,A -85,B 0,C 180,E1 -24958.075,E2 -24958.075} C_VEL
LIN {X 0,Y 139.637,Z 603.723,A -85,B 0,C 180,E1 -24963.616,E2 -24963.616} C_VEL
LIN {X 0,Y 146.139,Z 595.866,A -85,B 0,C 180,E1 -24968.694,E2 -24968.694} C_VEL
LIN {X 0,Y 152.43,Z 587.586,A -85,B 0,C 180,E1 -24972.797,E2 -24972.797} C_VEL
LIN {X 0,Y 159.688,Z 577.457,A -85,B 0,C 180,E1 -24976.565,E2 -24976.565} C_VEL
LIN {X 0,Y 166.355,Z 567.188,A -85,B 0,C 180,E1 -24979.501,E2 -24979.501} C_VEL
LIN {X 0,Y 173.599,Z 554.951,A -85,B 0,C 180,E1 -24982.131,E2 -24982.131} C_VEL
LIN {X 0,Y 179.915,Z 542.236,A -85,B 0,C 180,E1 -24984.305,E2 -24984.305} C_VEL
LIN {X 0,Y 185.488,Z 529.286,A -85,B 0,C 180,E1 -24985.976,E2 -24985.976} C_VEL
LIN {X 0,Y 190.818,Z 514.517,A -85,B 0,C 180,E1 -24987.403,E2 -24987.403} C_VEL
LIN {X 0,Y 194.906,Z 500.203,A -85,B 0,C 180,E1 -24988.414,E2 -24988.414} C_VEL
LIN {X 0,Y 198.221,Z 484.331,A -85,B 0,C 180,E1 -24989.227,E2 -24989.227} C_VEL
LIN {X 0,Y 200.347,Z 468.307,A -85,B 0,C 180,E1 -24989.744,E2 -24989.744} C_VEL
LIN {X 0,Y 204.676,Z 418.945,A -85,B 0,C 180,E1 -24991.056,E2 -24991.056} C_VEL
LIN {X 0,Y 201.41,Z 410.102,A -85,B 0,C 180,E1 -24993.444,E2 -24993.444} C_VEL
LIN {X 0,Y 197.952,Z 401.675,A -85,B 0,C 180,E1 -24996.227,E2 -24996.227} C_VEL
LIN {X 0,Y 195.772,Z 397.127,A -85,B 0,C 180,E1 -24998.133,E2 -24998.133} C_VEL
LIN {X 0,Y 191.74,Z 390.279,A -85,B 0,C 180,E1 -25002.113,E2 -25002.113} C_VEL
LIN {X 0,Y 188.908,Z 385.865,A -85,B 0,C 180,E1 -25005.594,E2 -25005.594} C_VEL
LIN {X 0,Y 186.579,Z 381.894,A -85,B 0,C 180,E1 -25009.419,E2 -25009.419} C_VEL
LIN {X 0,Y 184.707,Z 379.085,A -85,B 0,C 180,E1 -25013.994,E2 -25013.994} C_VEL
LIN {X 0,Y 184.187,Z 377.241,A -85,B 0,C 180,E1 -25016.719,E2 -25016.719} C_VEL
LIN {X 0,Y 183.882,Z 376.933,A -85,B 0,C 180,E1 -25020,E2 -25020} C_VEL
LIN {X 0,Y 184.271,Z 377.434,A -85,B 0,C 180,E1 -25024.238,E2 -25024.238} C_VEL
LIN {X 0,Y 185.683,Z 381.009,A -85,B 0,C 180,E1 -25029.257,E2 -25029.257} C_VEL
LIN {X 0,Y 186.862,Z 382.444,A -85,B 0,C 180,E1 -25031.58,E2 -25031.58} C_VEL
LIN {X 0,Y 189.179,Z 386.188,A -85,B 0,C 180,E1 -25035.211,E2 -25035.211} C_VEL
LIN {X 0,Y 192.342,Z 391.392,A -85,B 0,C 180,E1 -25039.001,E2 -25039.001} C_VEL
LIN {X 0,Y 194.937,Z 395.793,A -85,B 0,C 180,E1 -25041.57,E2 -25041.57} C_VEL
LIN {X 0,Y 199.131,Z 403.2,A -85,B 0,C 180,E1 -25045.1,E2 -25045.1} C_VEL
LIN {X 0,Y 203.585,Z 412.081,A -85,B 0,C 180,E1 -25048.338,E2 -25048.338} C_VEL
LIN {X 0,Y 204.928,Z 414.947,A -85,B 0,C 180,E1 -25049.236,E2 -25049.236} C_VEL
LIN {X 0,Y 199.996,Z 469.971,A -85,B 0,C 180,E1 -25050.745,E2 -25050.745} C_VEL
LIN {X 0,Y 197.347,Z 485.872,A -85,B 0,C 180,E1 -25051.399,E2 -25051.399} C_VEL
LIN {X 0,Y 193.583,Z 501.714,A -85,B 0,C 180,E1 -25052.428,E2 -25052.428} C_VEL
LIN {X 0,Y 189.448,Z 515.134,A -85,B 0,C 180,E1 -25053.612,E2 -25053.612} C_VEL
LIN {X 0,Y 184.252,Z 529.024,A -85,B 0,C 180,E1 -25055.256,E2 -25055.256} C_VEL
LIN {X 0,Y 177.894,Z 542.859,A -85,B 0,C 180,E1 -25057.34,E2 -25057.34} C_VEL
LIN {X 0,Y 171.324,Z 555.056,A -85,B 0,C 180,E1 -25059.724,E2 -25059.724} C_VEL
LIN {X 0,Y 164.491,Z 566.169,A -85,B 0,C 180,E1 -25062.524,E2 -25062.524} C_VEL
LIN {X 0,Y 158.134,Z 575.546,A -85,B 0,C 180,E1 -25065.6,E2 -25065.6} C_VEL
LIN {X 0,Y 152.319,Z 583.462,A -85,B 0,C 180,E1 -25068.892,E2 -25068.892} C_VEL
LIN {X 0,Y 145.239,Z 592.31,A -85,B 0,C 180,E1 -25073.648,E2 -25073.648} C_VEL
LIN {X 0,Y 139.836,Z 598.635,A -85,B 0,C 180,E1 -25078.15,E2 -25078.15} C_VEL
LIN {X 0,Y 134.839,Z 604.434,A -85,B 0,C 180,E1 -25083.703,E2 -25083.703} C_VEL
LIN {X 0,Y 131.792,Z 607.867,A -85,B 0,C 180,E1 -25088.082,E2 -25088.082} C_VEL
LIN {X 0,Y 128.943,Z 611.331,A -85,B 0,C 180,E1 -25094.186,E2 -25094.186} C_VEL
LIN {X 0,Y 127.194,Z 613.615,A -85,B 0,C 180,E1 -25100.459,E2 -25100.459} C_VEL
LIN {X 0,Y 126.513,Z 614.771,A -85,B 0,C 180,E1 -25106.816,E2 -25106.816} C_VEL
LIN {X 0,Y 126.505,Z 614.924,A -85,B 0,C 180,E1 -25110,E2 -25110} C_VEL
LIN {X 0,Y 126.743,Z 614.363,A -85,B 0,C 180,E1 -25116.367,E2 -25116.367} C_VEL
LIN {X 0,Y 127.913,Z 612.691,A -85,B 0,C 180,E1 -25122.695,E2 -25122.695} C_VEL
LIN {X 0,Y 130.135,Z 609.866,A -85,B 0,C 180,E1 -25128.906,E2 -25128.906} C_VEL
LIN {X 0,Y 133.752,Z 605.809,A -85,B 0,C 180,E1 -25134.857,E2 -25134.857} C_VEL
LIN {X 0,Y 138.468,Z 600.427,A -85,B 0,C 180,E1 -25140.5,E2 -25140.5} C_VEL
LIN {X 0,Y 144.339,Z 593.563,A -85,B 0,C 180,E1 -25145.752,E2 -25145.752} C_VEL
LIN {X 0,Y 151.275,Z 584.988,A -85,B 0,C 180,E1 -25150.572,E2 -25150.572} C_VEL
LIN {X 0,Y 156.009,Z 578.808,A -85,B 0,C 180,E1 -25153.266,E2 -25153.266} C_VEL
LIN {X 0,Y 161.176,Z 571.423,A -85,B 0,C 180,E1 -25156.009,E2 -25156.009} C_VEL
LIN {X 0,Y 167.815,Z 561.284,A -85,B 0,C 180,E1 -25158.922,E2 -25158.922} C_VEL
LIN {X 0,Y 174.743,Z 549.208,A -85,B 0,C 180,E1 -25161.651,E2 -25161.651} C_VEL
LIN {X 0,Y 180.877,Z 537.086,A -85,B 0,C 180,E1 -25163.729,E2 -25163.729} C_VEL
LIN {X 0,Y 186.556,Z 523.589,A -85,B 0,C 180,E1 -25165.592,E2 -25165.592} C_VEL
LIN {X 0,Y 191.552,Z 509.359,A -85,B 0,C 180,E1 -25167.062,E2 -25167.062} C_VEL
LIN {X 0,Y 195.462,Z 495.312,A -85,B 0,C 180,E1 -25168.15,E2 -25168.15} C_VEL
LIN {X 0,Y 198.567,Z 480.422,A -85,B 0,C 180,E1 -25168.988,E2 -25168.988} C_VEL
LIN {X 0,Y 200.635,Z 465.803,A -85,B 0,C 180,E1 -25169.524,E2 -25169.524} C_VEL
LIN {X 0,Y 205.131,Z 415.099,A -85,B 0,C 180,E1 -25170.89,E2 -25170.89} C_VEL
LIN {X 0,Y 200.921,Z 406.41,A -85,B 0,C 180,E1 -25173.828,E2 -25173.828} C_VEL
LIN {X 0,Y 197.258,Z 399.636,A -85,B 0,C 180,E1 -25176.711,E2 -25176.711} C_VEL
LIN {X 0,Y 193.826,Z 393.604,A -85,B 0,C 180,E1 -25179.85,E2 -25179.85} C_VEL
LIN {X 0,Y 191.338,Z 389.616,A -85,B 0,C 180,E1 -25182.498,E2 -25182.498} C_VEL
LIN {X 0,Y 189.216,Z 386.087,A -85,B 0,C 180,E1 -25185.205,E2 -25185.205} C_VEL
LIN {X 0,Y 187.215,Z 382.919,A -85,B 0,C 180,E1 -25188.359,E2 -25188.359} C_VEL
LIN {X 0,Y 186.813,Z 382.054,A -85,B 0,C 180,E1 -25189.158,E2 -25189.158} C_VEL
LIN {X 0,Y 184.958,Z 379.431,A -85,B 0,C 180,E1 -25193.716,E2 -25193.716} C_VEL
LIN {X 0,Y 184.437,Z 377.328,A -85,B 0,C 180,E1 -25196.723,E2 -25196.723} C_VEL
LIN {X 0,Y 184.339,Z 377.211,A -85,B 0,C 180,E1 -25202.185,E2 -25202.185} C_VEL
LIN {X 0,Y 184.509,Z 377.727,A -85,B 0,C 180,E1 -25203.548,E2 -25203.548} C_VEL
LIN {X 0,Y 186.167,Z 381.447,A -85,B 0,C 180,E1 -25209.232,E2 -25209.232} C_VEL
LIN {X 0,Y 186.988,Z 382.391,A -85,B 0,C 180,E1 -25210.832,E2 -25210.832} C_VEL
LIN {X 0,Y 189.838,Z 387.177,A -85,B 0,C 180,E1 -25215.294,E2 -25215.294} C_VEL
LIN {X 0,Y 192.48,Z 391.464,A -85,B 0,C 180,E1 -25218.416,E2 -25218.416} C_VEL
LIN {X 0,Y 195.269,Z 396.154,A -85,B 0,C 180,E1 -25221.182,E2 -25221.182} C_VEL
LIN {X 0,Y 197.242,Z 399.794,A -85,B 0,C 180,E1 -25222.935,E2 -25222.935} C_VEL
LIN {X 0,Y 200.865,Z 408.329,A -85,B 0,C 180,E1 -25225.935,E2 -25225.935} C_VEL
LIN {X 0,Y 204.808,Z 418.895,A -85,B 0,C 180,E1 -25228.859,E2 -25228.859} C_VEL
LIN {X 0,Y 199.683,Z 476.433,A -85,B 0,C 180,E1 -25230.467,E2 -25230.467} C_VEL
LIN {X 0,Y 196.955,Z 492.111,A -85,B 0,C 180,E1 -25231.088,E2 -25231.088} C_VEL
LIN {X 0,Y 193.218,Z 507.334,A -85,B 0,C 180,E1 -25232.013,E2 -25232.013} C_VEL
LIN {X 0,Y 188.833,Z 521.057,A -85,B 0,C 180,E1 -25233.135,E2 -25233.135} C_VEL
LIN {X 0,Y 183.567,Z 534.504,A -85,B 0,C 180,E1 -25234.602,E2 -25234.602} C_VEL
LIN {X 0,Y 178.066,Z 546.444,A -85,B 0,C 180,E1 -25236.301,E2 -25236.301} C_VEL
LIN {X 0,Y 171.775,Z 558.47,A -85,B 0,C 180,E1 -25238.514,E2 -25238.514} C_VEL
LIN {X 0,Y 165.234,Z 569.23,A -85,B 0,C 180,E1 -25240.979,E2 -25240.979} C_VEL
LIN {X 0,Y 158.611,Z 579.196,A -85,B 0,C 180,E1 -25243.945,E2 -25243.945} C_VEL
LIN {X 0,Y 151.512,Z 588.935,A -85,B 0,C 180,E1 -25247.721,E2 -25247.721} C_VEL
LIN {X 0,Y 145.273,Z 597.107,A -85,B 0,C 180,E1 -25251.917,E2 -25251.917} C_VEL
LIN {X 0,Y 144.247,Z 598.334,A -85,B 0,C 180,E1 -25252.665,E2 -25252.665} C_VEL
LIN {X 0,Y 141.348,Z 601.231,A -85,B 0,C 180,E1 -25254.38,E2 -25254.38} C_VEL
LIN {X 0,Y 135.174,Z 605.545,A -85,B 0,C 180,E1 -25257.042,E2 -25257.042} C_VEL
LIN {X 0,Y 129.185,Z 609.401,A -85,B 0,C 180,E1 -25260.037,E2 -25260.037} C_VEL
LIN {X 0,Y 126.675,Z 611.472,A -85,B 0,C 180,E1 -25262.244,E2 -25262.244} C_VEL
LIN {X 0,Y 123.892,Z 614.715,A -85,B 0,C 180,E1 -25266.604,E2 -25266.604} C_VEL
LIN {X 0,Y 120.954,Z 618.261,A -85,B 0,C 180,E1 -25273.111,E2 -25273.111} C_VEL
LIN {X 0,Y 119.503,Z 620.607,A -85,B 0,C 180,E1 -25279.838,E2 -25279.838} C_VEL
LIN {X 0,Y 119.182,Z 621.793,A -85,B 0,C 180,E1 -25286.619,E2 -25286.619} C_VEL
LIN {X 0,Y 119.332,Z 621.953,A -85,B 0,C 180,E1 -25290,E2 -25290} C_VEL
LIN {X 0,Y 119.204,Z 621.324,A -85,B 0,C 180,E1 -25296.772,E2 -25296.772} C_VEL
LIN {X 0,Y 120.046,Z 619.537,A -85,B 0,C 180,E1 -25303.543,E2 -25303.543} C_VEL
LIN {X 0,Y 122.236,Z 616.578,A -85,B 0,C 180,E1 -25310.179,E2 -25310.179} C_VEL
LIN {X 0,Y 125.693,Z 612.378,A -85,B 0,C 180,E1 -25316.571,E2 -25316.571} C_VEL
LIN {X 0,Y 130.742,Z 606.837,A -85,B 0,C 180,E1 -25322.516,E2 -25322.516} C_VEL
LIN {X 0,Y 137.075,Z 599.802,A -85,B 0,C 180,E1 -25327.969,E2 -25327.969} C_VEL
LIN {X 0,Y 143.39,Z 592.281,A -85,B 0,C 180,E1 -25332.37,E2 -25332.37} C_VEL
LIN {X 0,Y 150.439,Z 583.219,A -85,B 0,C 180,E1 -25336.393,E2 -25336.393} C_VEL
LIN {X 0,Y 158.321,Z 572.339,A -85,B 0,C 180,E1 -25339.971,E2 -25339.971} C_VEL
LIN {X 0,Y 165.508,Z 561.142,A -85,B 0,C 180,E1 -25342.765,E2 -25342.765} C_VEL
LIN {X 0,Y 171.798,Z 550.05,A -85,B 0,C 180,E1 -25344.9,E2 -25344.9} C_VEL
LIN {X 0,Y 178.263,Z 536.809,A -85,B 0,C 180,E1 -25346.904,E2 -25346.904} C_VEL
LIN {X 0,Y 183.635,Z 523.888,A -85,B 0,C 180,E1 -25348.377,E2 -25348.377} C_VEL
LIN {X 0,Y 188.49,Z 509.869,A -85,B 0,C 180,E1 -25349.566,E2 -25349.566} C_VEL
LIN {X 0,Y 192.51,Z 494.846,A -85,B 0,C 180,E1 -25350.51,E2 -25350.51} C_VEL
LIN {X 0,Y 195.451,Z 479.249,A -85,B 0,C 180,E1 -25351.199,E2 -25351.199} C_VEL
LIN {X 0,Y 197.727,Z 458.452,A -85,B 0,C 180,E1 -25351.787,E2 -25351.787} C_VEL
LIN {X 0,Y 201.037,Z 421.866,A -85,B 0,C 180,E1 -25352.749,E2 -25352.749} C_VEL
LIN {X 0,Y 197.69,Z 412.571,A -85,B 0,C 180,E1 -25355.455,E2 -25355.455} C_VEL
LIN {X 0,Y 194.502,Z 404.657,A -85,B 0,C 180,E1 -25358.332,E2 -25358.332} C_VEL
LIN {X 0,Y 191.163,Z 398.696,A -85,B 0,C 180,E1 -25361.652,E2 -25361.652} C_VEL
LIN {X 0,Y 189.392,Z 395.722,A -85,B 0,C 180,E1 -25363.702,E2 -25363.702} C_VEL
LIN {X 0,Y 187.515,Z 392.491,A -85,B 0,C 180,E1 -25366.255,E2 -25366.255} C_VEL
LIN {X 0,Y 185.428,Z 388.752,A -85,B 0,C 180,E1 -25369.904,E2 -25369.904} C_VEL
LIN {X 0,Y 183.658,Z 385.822,A -85,B 0,C 180,E1 -25374.648,E2 -25374.648} C_VEL
LIN {X 0,Y 183.318,Z 384.329,A -85,B 0,C 180,E1 -25376.704,E2 -25376.704} C_VEL
LIN {X 0,Y 183.016,Z 383.981,A -85,B 0,C 180,E1 -25380,E2 -25380} C_VEL
LIN {X 0,Y 183.363,Z 384.599,A -85,B 0,C 180,E1 -25384.121,E2 -25384.121} C_VEL
LIN {X 0,Y 184.813,Z 388.189,A -85,B 0,C 180,E1 -25389.301,E2 -25389.301} C_VEL
LIN {X 0,Y 185.685,Z 389.273,A -85,B 0,C 180,E1 -25391.075,E2 -25391.075} C_VEL
LIN {X 0,Y 188.28,Z 393.783,A -85,B 0,C 180,E1 -25395.286,E2 -25395.286} C_VEL
LIN {X 0,Y 190.737,Z 397.943,A -85,B 0,C 180,E1 -25398.322,E2 -25398.322} C_VEL
LIN {X 0,Y 193.947,Z 403.585,A -85,B 0,C 180,E1 -25401.597,E2 -25401.597} C_VEL
LIN {X 0,Y 197.53,Z 410.477,A -85,B 0,C 180,E1 -25404.712,E2 -25404.712} C_VEL
LIN {X 0,Y 201.272,Z 418.28,A -85,B 0,C 180,E1 -25407.555,E2 -25407.555} C_VEL
LIN {X 0,Y 196.451,Z 470.342,A -85,B 0,C 180,E1 -25408.974,E2 -25408.974} C_VEL
LIN {X 0,Y 193.753,Z 486.085,A -85,B 0,C 180,E1 -25409.612,E2 -25409.612} C_VEL
LIN {X 0,Y 189.882,Z 501.924,A -85,B 0,C 180,E1 -25410.626,E2 -25410.626} C_VEL
LIN {X 0,Y 185.226,Z 516.418,A -85,B 0,C 180,E1 -25411.903,E2 -25411.903} C_VEL
LIN {X 0,Y 180.135,Z 529.484,A -85,B 0,C 180,E1 -25413.444,E2 -25413.444} C_VEL
